SPLINE
SPL {X  -162.820, Y  +508.314, Z    +0.000, E1   +58.337, E3 +257283.169}
SPL {X  -162.820, Y  +498.518, Z    +0.000, E1   +58.346, E3 +257295.675}
SPL {X  -162.820, Y  +487.033, Z    +0.000, E1   +58.385, E3 +257310.273}
SPL {X  -162.820, Y  +474.470, Z    +0.000, E1   +58.318, E3 +257326.839}
SPL {X  -162.820, Y  +463.661, Z    +0.000, E1   +58.370, E3 +257340.278}
SPL {X  -162.820, Y  +454.904, Z    +0.000, E1   +58.380, E3 +257351.444}
SPL {X  -162.820, Y  +446.206, Z    +0.000, E1   +58.278, E3 +257363.335}
SPL {X  -162.820, Y  +436.416, Z    +0.000, E1   +58.325, E3 +257375.575}
SPL {X  -162.820, Y  +426.628, Z    +0.000, E1   +58.432, E3 +257387.443}
SPL {X  -162.820, Y  +415.377, Z    +0.000, E1   +58.239, E3 +257403.375}
SPL {X  -162.820, Y  +403.663, Z    +0.000, E1   +58.258, E3 +257418.154}
SPL {X  -162.820, Y  +397.157, Z    +0.000, E1   +58.054, E3 +257427.890}
SPL {X  -162.820, Y  +387.359, Z    +0.000, E1   +58.365, E3 +257438.519}
SPL {X  -162.810, Y  +378.731, Z    +0.000, E1   +58.366, E3 +257449.577}
SPL {X  -162.546, Y  +371.051, Z    +0.000, E1   +58.239, E3 +257460.297}
SPL {X  -161.863, Y  +362.875, Z    +0.000, E1   +58.273, E3 +257470.522}
SPL {X  -161.159, Y  +357.301, Z    +0.000, E1   +57.946, E3 +257479.822}
SPL {X  -159.864, Y  +349.614, Z    +0.000, E1   +57.922, E3 +257489.898}
SPL {X  -158.548, Y  +343.449, Z    +0.000, E1   +57.711, E3 +257499.072}
SPL {X  -156.580, Y  +335.856, Z    +0.000, E1   +57.340, E3 +257511.295}
SPL {X  -154.237, Y  +328.333, Z    +0.000, E1   +56.930, E3 +257523.214}
SPL {X  -152.732, Y  +324.078, Z    +0.000, E1   +56.482, E3 +257531.219}
SPL {X  -150.609, Y  +318.634, Z    +0.000, E1   +56.366, E3 +257538.913}
SPL {X  -148.206, Y  +313.080, Z    +0.000, E1   +55.888, E3 +257548.625}
SPL {X  -145.956, Y  +308.339, Z    +0.000, E1   +55.380, E3 +257557.301}
SPL {X  -143.330, Y  +303.254, Z    +0.000, E1   +55.057, E3 +257565.421}
SPL {X  -137.431, Y  +293.190, Z    +0.000, E1   +56.809, E3 +257569.584}
SPL {X  -115.845, Y  +266.087, Z    +0.000, E1   +50.276, E3 +257668.442}
SPL {X  -114.083, Y  +264.330, Z    +0.000, E1   +49.123, E3 +257707.152}
ENDSPLINE

SPLINE
SPL {X  -149.622, Y  +316.285, Z    +0.000, E1   +35.036, E3 +257775.664}
SPL {X  -158.704, Y  +344.121, Z    +0.000, E1   +23.312, E3 +257785.537}
SPL {X  -162.109, Y  +365.304, Z    +0.000, E1   +11.761, E3 +257784.839}
SPL {X  -162.811, Y  +378.776, Z    +0.000, E1    +3.078, E3 +257785.083}
SPL {X  -162.820, Y  +382.545, Z    +0.000, E1    +0.100, E3 +257784.644}
SPL {X  -162.820, Y  +384.317, Z    +0.000, E1    -1.618, E3 +257784.463}
SPL {X  -162.820, Y  +387.033, Z    +0.000, E1    -4.758, E3 +257784.255}
SPL {X  -162.820, Y  +390.967, Z    +0.000, E1    -9.918, E3 +257784.700}
SPL {X  -162.820, Y  +397.718, Z    +0.000, E1   -19.761, E3 +257784.074}
SPL {X  -162.820, Y  +405.058, Z    +0.000, E1   -29.962, E3 +257784.987}
SPL {X  -162.820, Y  +417.515, Z    +0.000, E1   -44.878, E3 +257784.149}
SPL {X  -162.820, Y  +462.065, Z    +0.000, E1   -61.507, E3 +257801.109}
SPL {X  -162.820, Y  +504.602, Z    +0.000, E1   -64.286, E3 +257826.635}
SPL {X  -162.820, Y  +535.709, Z    +0.000, E1   -59.182, E3 +257884.314}
SPL {X  -162.820, Y  +543.678, Z    +0.000, E1   -58.515, E3 +257898.703}
SPL {X  -162.820, Y  +553.725, Z    +0.000, E1   -58.454, E3 +257911.964}
SPL {X  -162.820, Y  +562.850, Z    +0.000, E1   -58.373, E3 +257924.126}
SPL {X  -162.820, Y  +571.217, Z    +0.000, E1   -58.397, E3 +257934.679}
SPL {X  -162.820, Y  +581.879, Z    +0.000, E1   -58.475, E3 +257947.932}
SPL {X  -162.820, Y  +591.768, Z    +0.000, E1   -58.375, E3 +257961.130}
SPL {X  -162.820, Y  +601.090, Z    +0.000, E1   -58.519, E3 +257972.117}
SPL {X  -162.820, Y  +609.492, Z    +0.000, E1   -58.431, E3 +257983.422}
SPL {X  -162.820, Y  +617.241, Z    +0.000, E1   -58.340, E3 +257993.947}
SPL {X  -162.820, Y  +626.506, Z    +0.000, E1   -58.420, E3 +258005.329}
SPL {X  -162.820, Y  +635.919, Z    +0.000, E1   -58.604, E3 +258016.073}
SPL {X  -162.820, Y  +643.895, Z    +0.000, E1   -58.380, E3 +258027.838}
SPL {X  -162.820, Y  +653.118, Z    +0.000, E1   -58.401, E3 +258039.435}
SPL {X  -162.820, Y  +660.924, Z    +0.000, E1   -58.393, E3 +258049.503}
SPL {X  -162.820, Y  +670.459, Z    +0.000, E1   -58.489, E3 +258061.104}
SPL {X  -162.713, Y  +679.396, Z    +0.000, E1   -58.414, E3 +258073.003}
SPL {X  -162.301, Y  +686.495, Z    +0.000, E1   -58.302, E3 +258082.787}
SPL {X  -161.571, Y  +693.631, Z    +0.000, E1   -58.186, E3 +258092.751}
SPL {X  -160.411, Y  +701.402, Z    +0.000, E1   -58.100, E3 +258103.227}
SPL {X  -159.229, Y  +707.508, Z    +0.000, E1   -57.870, E3 +258112.465}
SPL {X  -157.825, Y  +713.519, Z    +0.000, E1   -57.630, E3 +258121.701}
SPL {X  -156.079, Y  +719.864, Z    +0.000, E1   -57.324, E3 +258131.664}
SPL {X  -154.064, Y  +726.175, Z    +0.000, E1   -57.042, E3 +258141.426}
SPL {X  -152.053, Y  +731.726, Z    +0.000, E1   -56.648, E3 +258150.711}
SPL {X  -150.108, Y  +736.570, Z    +0.000, E1   -56.283, E3 +258158.950}
SPL {X  -147.726, Y  +741.964, Z    +0.000, E1   -55.884, E3 +258167.986}
SPL {X  -145.163, Y  +747.242, Z    +0.000, E1   -55.517, E3 +258176.582}
SPL {X  -142.489, Y  +752.286, Z    +0.000, E1   -55.227, E3 +258184.409}
SPL {X  -136.074, Y  +762.910, Z    +0.000, E1   -57.336, E3 +258187.531}
SPL {X  -116.561, Y  +787.183, Z    +0.000, E1   -51.088, E3 +258271.999}
ENDSPLINE

SPLINE
SPL {X  -119.623, Y  +783.957, Z    +0.000, E1   -49.202, E3 +258396.532}
SPL {X  -149.958, Y  +736.927, Z    +0.000, E1   -34.772, E3 +258394.249}
SPL {X  -158.826, Y  +709.343, Z    +0.000, E1   -23.029, E3 +258402.592}
SPL {X  -161.800, Y  +691.694, Z    +0.000, E1   -13.520, E3 +258404.886}
SPL {X  -162.711, Y  +679.444, Z    +0.000, E1    -5.922, E3 +258404.960}
SPL {X  -162.820, Y  +673.886, Z    +0.000, E1    -1.998, E3 +258405.121}
SPL {X  -162.820, Y  +671.620, Z    +0.000, E1    -0.225, E3 +258404.696}
SPL {X  -162.820, Y  +669.030, Z    +0.000, E1    +2.242, E3 +258404.397}
SPL {X  -162.820, Y  +664.667, Z    +0.000, E1    +7.867, E3 +258404.100}
SPL {X  -162.820, Y  +660.022, Z    +0.000, E1   +14.535, E3 +258403.997}
SPL {X  -162.820, Y  +653.408, Z    +0.000, E1   +24.221, E3 +258404.307}
SPL {X  -162.820, Y  +640.244, Z    +0.000, E1   +41.042, E3 +258404.351}
SPL {X  -162.820, Y  +592.517, Z    +0.000, E1   +60.575, E3 +258423.482}
SPL {X  -162.820, Y  +515.613, Z    +0.000, E1   +60.751, E3 +258497.317}
ENDSPLINE

SPLINE
SPL {X  -162.820, Y  +518.198, Z    +0.000, E1   +58.338, E3 +258510.473}
ENDSPLINE

SPLINE
SPL {X  -162.820, Y  +508.314, Z    +0.000, E1   +58.337, E3 +258523.169}
SPL {X  -162.820, Y  +498.518, Z    +0.000, E1   +58.346, E3 +258535.675}
SPL {X  -162.820, Y  +489.418, Z    +0.000, E1   +58.357, E3 +258547.265}
SPL {X  -162.820, Y  +479.904, Z    +0.000, E1   +58.389, E3 +258559.312}
SPL {X  -162.820, Y  +472.095, Z    +0.000, E1   +58.202, E3 +258570.492}
SPL {X  -162.820, Y  +463.661, Z    +0.000, E1   +58.370, E3 +258580.278}
SPL {X  -162.820, Y  +454.904, Z    +0.000, E1   +58.380, E3 +258591.444}
SPL {X  -162.820, Y  +446.206, Z    +0.000, E1   +58.278, E3 +258603.335}
SPL {X  -162.820, Y  +436.416, Z    +0.000, E1   +58.325, E3 +258615.575}
SPL {X  -162.820, Y  +426.628, Z    +0.000, E1   +58.432, E3 +258627.443}
SPL {X  -162.820, Y  +418.389, Z    +0.000, E1   +58.300, E3 +258638.846}
SPL {X  -162.820, Y  +412.292, Z    +0.000, E1   +58.070, E3 +258648.214}
SPL {X  -162.820, Y  +403.663, Z    +0.000, E1   +58.258, E3 +258658.154}
SPL {X  -162.820, Y  +397.157, Z    +0.000, E1   +58.054, E3 +258667.890}
SPL {X  -162.820, Y  +387.359, Z    +0.000, E1   +58.365, E3 +258678.519}
SPL {X  -162.810, Y  +378.731, Z    +0.000, E1   +58.366, E3 +258689.577}
SPL {X  -162.546, Y  +371.051, Z    +0.000, E1   +58.239, E3 +258700.297}
SPL {X  -161.863, Y  +362.875, Z    +0.000, E1   +58.273, E3 +258710.522}
SPL {X  -161.159, Y  +357.301, Z    +0.000, E1   +57.946, E3 +258719.822}
SPL {X  -159.864, Y  +349.614, Z    +0.000, E1   +57.922, E3 +258729.898}
SPL {X  -158.548, Y  +343.449, Z    +0.000, E1   +57.711, E3 +258739.072}
SPL {X  -156.580, Y  +335.856, Z    +0.000, E1   +57.340, E3 +258751.295}
SPL {X  -154.237, Y  +328.333, Z    +0.000, E1   +56.930, E3 +258763.214}
SPL {X  -152.732, Y  +324.078, Z    +0.000, E1   +56.482, E3 +258771.219}
SPL {X  -150.609, Y  +318.634, Z    +0.000, E1   +56.366, E3 +258778.913}
SPL {X  -148.206, Y  +313.080, Z    +0.000, E1   +55.888, E3 +258788.625}
SPL {X  -145.956, Y  +308.339, Z    +0.000, E1   +55.380, E3 +258797.301}
SPL {X  -143.330, Y  +303.254, Z    +0.000, E1   +55.057, E3 +258805.421}
SPL {X  -137.431, Y  +293.190, Z    +0.000, E1   +56.809, E3 +258809.584}
SPL {X  -115.845, Y  +266.087, Z    +0.000, E1   +50.276, E3 +258908.442}
SPL {X  -114.083, Y  +264.330, Z    +0.000, E1   +49.123, E3 +258947.152}
ENDSPLINE

SPLINE
SPL {X  -149.622, Y  +316.285, Z    +0.000, E1   +35.036, E3 +259015.664}
SPL {X  -158.704, Y  +344.121, Z    +0.000, E1   +23.312, E3 +259025.537}
SPL {X  -162.109, Y  +365.304, Z    +0.000, E1   +11.761, E3 +259024.839}
SPL {X  -162.811, Y  +378.776, Z    +0.000, E1    +3.078, E3 +259025.083}
SPL {X  -162.820, Y  +383.454, Z    +0.000, E1    -0.619, E3 +259024.551}
SPL {X  -162.820, Y  +387.033, Z    +0.000, E1    -4.758, E3 +259024.255}
SPL {X  -162.820, Y  +390.967, Z    +0.000, E1    -9.918, E3 +259024.700}
SPL {X  -162.820, Y  +397.718, Z    +0.000, E1   -19.761, E3 +259024.074}
SPL {X  -162.820, Y  +405.058, Z    +0.000, E1   -29.962, E3 +259024.987}
SPL {X  -162.820, Y  +417.515, Z    +0.000, E1   -44.878, E3 +259024.149}
SPL {X  -162.820, Y  +462.065, Z    +0.000, E1   -61.507, E3 +259041.109}
SPL {X  -162.820, Y  +504.602, Z    +0.000, E1   -64.286, E3 +259066.635}
SPL {X  -162.820, Y  +535.709, Z    +0.000, E1   -59.182, E3 +259124.314}
SPL {X  -162.820, Y  +543.678, Z    +0.000, E1   -58.515, E3 +259138.703}
SPL {X  -162.820, Y  +553.725, Z    +0.000, E1   -58.454, E3 +259151.964}
SPL {X  -162.820, Y  +562.850, Z    +0.000, E1   -58.373, E3 +259164.126}
SPL {X  -162.820, Y  +573.452, Z    +0.000, E1   -58.444, E3 +259177.339}
SPL {X  -162.820, Y  +583.632, Z    +0.000, E1   -58.444, E3 +259190.266}
SPL {X  -162.820, Y  +591.768, Z    +0.000, E1   -58.375, E3 +259201.130}
SPL {X  -162.820, Y  +601.090, Z    +0.000, E1   -58.519, E3 +259212.117}
SPL {X  -162.820, Y  +609.492, Z    +0.000, E1   -58.431, E3 +259223.422}
SPL {X  -162.820, Y  +617.241, Z    +0.000, E1   -58.340, E3 +259233.947}
SPL {X  -162.820, Y  +626.506, Z    +0.000, E1   -58.420, E3 +259245.329}
SPL {X  -162.820, Y  +635.919, Z    +0.000, E1   -58.604, E3 +259256.073}
SPL {X  -162.820, Y  +643.895, Z    +0.000, E1   -58.380, E3 +259267.838}
SPL {X  -162.820, Y  +653.118, Z    +0.000, E1   -58.401, E3 +259279.435}
SPL {X  -162.820, Y  +660.924, Z    +0.000, E1   -58.393, E3 +259289.503}
SPL {X  -162.820, Y  +670.459, Z    +0.000, E1   -58.489, E3 +259301.104}
SPL {X  -162.713, Y  +679.396, Z    +0.000, E1   -58.414, E3 +259313.003}
SPL {X  -162.301, Y  +686.495, Z    +0.000, E1   -58.302, E3 +259322.787}
SPL {X  -161.571, Y  +693.631, Z    +0.000, E1   -58.186, E3 +259332.751}
SPL {X  -160.411, Y  +701.402, Z    +0.000, E1   -58.100, E3 +259343.227}
SPL {X  -159.229, Y  +707.508, Z    +0.000, E1   -57.870, E3 +259352.465}
SPL {X  -157.825, Y  +713.519, Z    +0.000, E1   -57.630, E3 +259361.701}
SPL {X  -156.079, Y  +719.864, Z    +0.000, E1   -57.324, E3 +259371.664}
SPL {X  -154.064, Y  +726.175, Z    +0.000, E1   -57.042, E3 +259381.426}
SPL {X  -152.053, Y  +731.726, Z    +0.000, E1   -56.648, E3 +259390.711}
SPL {X  -150.108, Y  +736.570, Z    +0.000, E1   -56.283, E3 +259398.950}
SPL {X  -147.726, Y  +741.964, Z    +0.000, E1   -55.884, E3 +259407.986}
SPL {X  -145.163, Y  +747.242, Z    +0.000, E1   -55.517, E3 +259416.582}
SPL {X  -142.489, Y  +752.286, Z    +0.000, E1   -55.227, E3 +259424.409}
SPL {X  -136.074, Y  +762.910, Z    +0.000, E1   -57.336, E3 +259427.531}
SPL {X  -116.561, Y  +787.183, Z    +0.000, E1   -51.088, E3 +259511.999}
ENDSPLINE

SPLINE
SPL {X  -119.623, Y  +783.957, Z    +0.000, E1   -49.202, E3 +259636.532}
SPL {X  -149.958, Y  +736.927, Z    +0.000, E1   -34.772, E3 +259634.249}
SPL {X  -158.826, Y  +709.343, Z    +0.000, E1   -23.029, E3 +259642.592}
SPL {X  -161.800, Y  +691.694, Z    +0.000, E1   -13.520, E3 +259644.886}
SPL {X  -162.711, Y  +679.444, Z    +0.000, E1    -5.922, E3 +259644.960}
SPL {X  -162.820, Y  +672.303, Z    +0.000, E1    -0.875, E3 +259644.825}
SPL {X  -162.820, Y  +669.030, Z    +0.000, E1    +2.242, E3 +259644.397}
SPL {X  -162.820, Y  +664.667, Z    +0.000, E1    +7.867, E3 +259644.100}
SPL {X  -162.820, Y  +660.022, Z    +0.000, E1   +14.535, E3 +259643.997}
SPL {X  -162.820, Y  +653.408, Z    +0.000, E1   +24.221, E3 +259644.307}
SPL {X  -162.820, Y  +640.244, Z    +0.000, E1   +41.042, E3 +259644.351}
SPL {X  -162.820, Y  +592.517, Z    +0.000, E1   +60.575, E3 +259663.482}
SPL {X  -162.820, Y  +515.613, Z    +0.000, E1   +60.751, E3 +259737.317}
ENDSPLINE

SPLINE
SPL {X  -162.820, Y  +518.198, Z    +0.000, E1   +58.338, E3 +259750.473}
ENDSPLINE

SPLINE
SPL {X  -162.820, Y  +508.314, Z    +0.000, E1   +58.337, E3 +259763.169}
SPL {X  -162.820, Y  +498.518, Z    +0.000, E1   +58.346, E3 +259775.675}
SPL {X  -162.820, Y  +489.418, Z    +0.000, E1   +58.357, E3 +259787.265}
SPL {X  -162.820, Y  +479.904, Z    +0.000, E1   +58.389, E3 +259799.312}
SPL {X  -162.820, Y  +472.095, Z    +0.000, E1   +58.202, E3 +259810.492}
SPL {X  -162.820, Y  +463.661, Z    +0.000, E1   +58.370, E3 +259820.278}
SPL {X  -162.820, Y  +454.904, Z    +0.000, E1   +58.380, E3 +259831.444}
SPL {X  -162.820, Y  +446.206, Z    +0.000, E1   +58.278, E3 +259843.335}
SPL {X  -162.820, Y  +436.416, Z    +0.000, E1   +58.325, E3 +259855.575}
SPL {X  -162.820, Y  +426.628, Z    +0.000, E1   +58.432, E3 +259867.443}
SPL {X  -162.820, Y  +415.377, Z    +0.000, E1   +58.239, E3 +259883.375}
SPL {X  -162.820, Y  +403.663, Z    +0.000, E1   +58.258, E3 +259898.154}
SPL {X  -162.820, Y  +397.157, Z    +0.000, E1   +58.054, E3 +259907.890}
SPL {X  -162.820, Y  +387.359, Z    +0.000, E1   +58.365, E3 +259918.519}
SPL {X  -162.810, Y  +378.731, Z    +0.000, E1   +58.366, E3 +259929.577}
SPL {X  -162.546, Y  +371.051, Z    +0.000, E1   +58.239, E3 +259940.297}
SPL {X  -161.863, Y  +362.875, Z    +0.000, E1   +58.273, E3 +259950.522}
SPL {X  -161.159, Y  +357.301, Z    +0.000, E1   +57.946, E3 +259959.822}
SPL {X  -159.864, Y  +349.614, Z    +0.000, E1   +57.922, E3 +259969.898}
SPL {X  -158.548, Y  +343.449, Z    +0.000, E1   +57.711, E3 +259979.072}
SPL {X  -156.580, Y  +335.856, Z    +0.000, E1   +57.340, E3 +259991.295}
SPL {X  -154.237, Y  +328.333, Z    +0.000, E1   +56.930, E3 +260003.214}
SPL {X  -152.732, Y  +324.078, Z    +0.000, E1   +56.482, E3 +260011.219}
SPL {X  -150.609, Y  +318.634, Z    +0.000, E1   +56.366, E3 +260018.913}
SPL {X  -148.206, Y  +313.080, Z    +0.000, E1   +55.888, E3 +260028.625}
SPL {X  -145.956, Y  +308.339, Z    +0.000, E1   +55.380, E3 +260037.301}
SPL {X  -143.330, Y  +303.254, Z    +0.000, E1   +55.057, E3 +260045.421}
SPL {X  -137.431, Y  +293.190, Z    +0.000, E1   +56.809, E3 +260049.584}
SPL {X  -115.845, Y  +266.087, Z    +0.000, E1   +50.276, E3 +260148.442}
SPL {X  -114.083, Y  +264.330, Z    +0.000, E1   +49.123, E3 +260187.152}
ENDSPLINE

SPLINE
SPL {X  -149.622, Y  +316.285, Z    +0.000, E1   +35.036, E3 +260255.664}
SPL {X  -158.704, Y  +344.121, Z    +0.000, E1   +23.312, E3 +260265.537}
SPL {X  -161.701, Y  +361.440, Z    +0.000, E1   +13.961, E3 +260264.608}
SPL {X  -162.691, Y  +374.019, Z    +0.000, E1    +6.263, E3 +260265.261}
SPL {X  -162.820, Y  +381.771, Z    +0.000, E1    +0.850, E3 +260264.745}
SPL {X  -162.820, Y  +384.317, Z    +0.000, E1    -1.618, E3 +260264.463}
SPL {X  -162.820, Y  +387.033, Z    +0.000, E1    -4.758, E3 +260264.255}
SPL {X  -162.820, Y  +390.967, Z    +0.000, E1    -9.918, E3 +260264.700}
SPL {X  -162.820, Y  +395.392, Z    +0.000, E1   -16.726, E3 +260263.141}
SPL {X  -162.820, Y  +402.654, Z    +0.000, E1   -26.492, E3 +260265.032}
SPL {X  -162.820, Y  +417.515, Z    +0.000, E1   -44.878, E3 +260264.149}
SPL {X  -162.820, Y  +462.065, Z    +0.000, E1   -61.507, E3 +260281.109}
SPL {X  -162.820, Y  +504.602, Z    +0.000, E1   -64.286, E3 +260306.635}
SPL {X  -162.820, Y  +535.709, Z    +0.000, E1   -59.182, E3 +260364.314}
SPL {X  -162.820, Y  +543.678, Z    +0.000, E1   -58.515, E3 +260378.703}
SPL {X  -162.820, Y  +553.725, Z    +0.000, E1   -58.454, E3 +260391.964}
SPL {X  -162.820, Y  +562.850, Z    +0.000, E1   -58.373, E3 +260404.126}
SPL {X  -162.820, Y  +571.217, Z    +0.000, E1   -58.397, E3 +260414.679}
SPL {X  -162.820, Y  +581.879, Z    +0.000, E1   -58.475, E3 +260427.932}
SPL {X  -162.820, Y  +591.768, Z    +0.000, E1   -58.375, E3 +260441.130}
SPL {X  -162.820, Y  +601.090, Z    +0.000, E1   -58.519, E3 +260452.117}
SPL {X  -162.820, Y  +609.492, Z    +0.000, E1   -58.431, E3 +260463.422}
SPL {X  -162.820, Y  +617.241, Z    +0.000, E1   -58.340, E3 +260473.947}
SPL {X  -162.820, Y  +626.506, Z    +0.000, E1   -58.420, E3 +260485.329}
SPL {X  -162.820, Y  +635.919, Z    +0.000, E1   -58.604, E3 +260496.073}
SPL {X  -162.820, Y  +643.895, Z    +0.000, E1   -58.380, E3 +260507.838}
SPL {X  -162.820, Y  +653.118, Z    +0.000, E1   -58.401, E3 +260519.435}
SPL {X  -162.820, Y  +660.924, Z    +0.000, E1   -58.393, E3 +260529.503}
SPL {X  -162.820, Y  +670.459, Z    +0.000, E1   -58.489, E3 +260541.104}
SPL {X  -162.713, Y  +679.396, Z    +0.000, E1   -58.414, E3 +260553.003}
SPL {X  -162.301, Y  +686.495, Z    +0.000, E1   -58.302, E3 +260562.787}
SPL {X  -161.571, Y  +693.631, Z    +0.000, E1   -58.186, E3 +260572.751}
SPL {X  -160.411, Y  +701.402, Z    +0.000, E1   -58.100, E3 +260583.227}
SPL {X  -159.229, Y  +707.508, Z    +0.000, E1   -57.870, E3 +260592.465}
SPL {X  -157.825, Y  +713.519, Z    +0.000, E1   -57.630, E3 +260601.701}
SPL {X  -156.079, Y  +719.864, Z    +0.000, E1   -57.324, E3 +260611.664}
SPL {X  -154.064, Y  +726.175, Z    +0.000, E1   -57.042, E3 +260621.426}
SPL {X  -152.053, Y  +731.726, Z    +0.000, E1   -56.648, E3 +260630.711}
SPL {X  -150.108, Y  +736.570, Z    +0.000, E1   -56.283, E3 +260638.950}
SPL {X  -147.726, Y  +741.964, Z    +0.000, E1   -55.884, E3 +260647.986}
SPL {X  -145.163, Y  +747.242, Z    +0.000, E1   -55.517, E3 +260656.582}
SPL {X  -142.489, Y  +752.286, Z    +0.000, E1   -55.227, E3 +260664.409}
SPL {X  -136.074, Y  +762.910, Z    +0.000, E1   -57.336, E3 +260667.531}
SPL {X  -116.561, Y  +787.183, Z    +0.000, E1   -51.088, E3 +260751.999}
ENDSPLINE

SPLINE
SPL {X  -119.623, Y  +783.957, Z    +0.000, E1   -49.202, E3 +260876.532}
SPL {X  -149.958, Y  +736.927, Z    +0.000, E1   -34.772, E3 +260874.249}
SPL {X  -158.826, Y  +709.343, Z    +0.000, E1   -23.029, E3 +260882.592}
SPL {X  -161.800, Y  +691.694, Z    +0.000, E1   -13.520, E3 +260884.886}
SPL {X  -162.711, Y  +679.444, Z    +0.000, E1    -5.922, E3 +260884.960}
SPL {X  -162.820, Y  +672.303, Z    +0.000, E1    -0.875, E3 +260884.825}
SPL {X  -162.820, Y  +669.030, Z    +0.000, E1    +2.242, E3 +260884.397}
SPL {X  -162.820, Y  +664.667, Z    +0.000, E1    +7.867, E3 +260884.100}
SPL {X  -162.820, Y  +660.022, Z    +0.000, E1   +14.535, E3 +260883.997}
SPL {X  -162.820, Y  +653.408, Z    +0.000, E1   +24.221, E3 +260884.307}
SPL {X  -162.820, Y  +640.244, Z    +0.000, E1   +41.042, E3 +260884.351}
SPL {X  -162.820, Y  +602.578, Z    +0.000, E1   +60.061, E3 +260895.766}
SPL {X  -162.820, Y  +586.468, Z    +0.000, E1   +60.779, E3 +260908.168}
SPL {X  -162.820, Y  +515.613, Z    +0.000, E1   +60.751, E3 +260977.317}
ENDSPLINE

SPLINE
SPL {X  -162.820, Y  +518.198, Z    +0.000, E1   +58.338, E3 +260990.473}
ENDSPLINE

SPLINE
SPL {X  -162.820, Y  +508.314, Z    +0.000, E1   +58.337, E3 +261003.169}
SPL {X  -162.820, Y  +498.518, Z    +0.000, E1   +58.346, E3 +261015.675}
SPL {X  -162.820, Y  +489.418, Z    +0.000, E1   +58.357, E3 +261027.265}
SPL {X  -162.820, Y  +479.904, Z    +0.000, E1   +58.389, E3 +261039.312}
SPL {X  -162.820, Y  +472.095, Z    +0.000, E1   +58.202, E3 +261050.492}
SPL {X  -162.820, Y  +463.661, Z    +0.000, E1   +58.370, E3 +261060.278}
SPL {X  -162.820, Y  +454.904, Z    +0.000, E1   +58.380, E3 +261071.444}
SPL {X  -162.820, Y  +446.206, Z    +0.000, E1   +58.278, E3 +261083.335}
SPL {X  -162.820, Y  +436.416, Z    +0.000, E1   +58.325, E3 +261095.575}
SPL {X  -162.820, Y  +426.628, Z    +0.000, E1   +58.432, E3 +261107.443}
SPL {X  -162.820, Y  +415.377, Z    +0.000, E1   +58.239, E3 +261123.375}
SPL {X  -162.820, Y  +403.663, Z    +0.000, E1   +58.258, E3 +261138.154}
SPL {X  -162.820, Y  +397.157, Z    +0.000, E1   +58.054, E3 +261147.890}
SPL {X  -162.820, Y  +387.359, Z    +0.000, E1   +58.365, E3 +261158.519}
SPL {X  -162.810, Y  +378.731, Z    +0.000, E1   +58.366, E3 +261169.577}
SPL {X  -162.546, Y  +371.051, Z    +0.000, E1   +58.239, E3 +261180.297}
SPL {X  -161.863, Y  +362.875, Z    +0.000, E1   +58.273, E3 +261190.522}
SPL {X  -161.159, Y  +357.301, Z    +0.000, E1   +57.946, E3 +261199.822}
SPL {X  -159.864, Y  +349.614, Z    +0.000, E1   +57.922, E3 +261209.898}
SPL {X  -158.548, Y  +343.449, Z    +0.000, E1   +57.711, E3 +261219.072}
SPL {X  -156.580, Y  +335.856, Z    +0.000, E1   +57.340, E3 +261231.295}
SPL {X  -154.237, Y  +328.333, Z    +0.000, E1   +56.930, E3 +261243.214}
SPL {X  -152.732, Y  +324.078, Z    +0.000, E1   +56.482, E3 +261251.219}
SPL {X  -150.609, Y  +318.634, Z    +0.000, E1   +56.366, E3 +261258.913}
SPL {X  -148.206, Y  +313.080, Z    +0.000, E1   +55.888, E3 +261268.625}
SPL {X  -145.956, Y  +308.339, Z    +0.000, E1   +55.380, E3 +261277.301}
SPL {X  -143.330, Y  +303.254, Z    +0.000, E1   +55.057, E3 +261285.421}
SPL {X  -137.431, Y  +293.190, Z    +0.000, E1   +56.809, E3 +261289.584}
SPL {X  -115.845, Y  +266.087, Z    +0.000, E1   +50.276, E3 +261388.442}
SPL {X  -114.083, Y  +264.330, Z    +0.000, E1   +49.123, E3 +261427.152}
ENDSPLINE

SPLINE
SPL {X  -136.188, Y  +291.263, Z    +0.000, E1   +45.457, E3 +261523.218}
SPL {X  -151.738, Y  +321.457, Z    +0.000, E1   +32.773, E3 +261490.387}
SPL {X  -158.704, Y  +344.121, Z    +0.000, E1   +23.312, E3 +261505.537}
SPL {X  -161.701, Y  +361.440, Z    +0.000, E1   +13.961, E3 +261504.608}
SPL {X  -162.691, Y  +374.019, Z    +0.000, E1    +6.263, E3 +261505.261}
SPL {X  -162.820, Y  +380.238, Z    +0.000, E1    +1.925, E3 +261504.945}
SPL {X  -162.820, Y  +382.545, Z    +0.000, E1    +0.100, E3 +261504.644}
SPL {X  -162.820, Y  +384.317, Z    +0.000, E1    -1.618, E3 +261504.463}
SPL {X  -162.820, Y  +387.033, Z    +0.000, E1    -4.758, E3 +261504.255}
SPL {X  -162.820, Y  +390.967, Z    +0.000, E1    -9.918, E3 +261504.700}
SPL {X  -162.820, Y  +395.392, Z    +0.000, E1   -16.726, E3 +261503.141}
SPL {X  -162.820, Y  +402.654, Z    +0.000, E1   -26.492, E3 +261505.032}
SPL {X  -162.820, Y  +417.515, Z    +0.000, E1   -44.878, E3 +261504.149}
SPL {X  -162.820, Y  +462.065, Z    +0.000, E1   -61.507, E3 +261521.109}
SPL {X  -162.820, Y  +504.602, Z    +0.000, E1   -64.286, E3 +261546.635}
SPL {X  -162.820, Y  +535.709, Z    +0.000, E1   -59.182, E3 +261604.314}
SPL {X  -162.820, Y  +543.678, Z    +0.000, E1   -58.515, E3 +261618.703}
SPL {X  -162.820, Y  +553.725, Z    +0.000, E1   -58.454, E3 +261631.964}
SPL {X  -162.820, Y  +562.850, Z    +0.000, E1   -58.373, E3 +261644.126}
SPL {X  -162.820, Y  +573.452, Z    +0.000, E1   -58.444, E3 +261657.339}
SPL {X  -162.820, Y  +583.632, Z    +0.000, E1   -58.444, E3 +261670.266}
SPL {X  -162.820, Y  +591.768, Z    +0.000, E1   -58.375, E3 +261681.130}
SPL {X  -162.820, Y  +601.090, Z    +0.000, E1   -58.519, E3 +261692.117}
SPL {X  -162.820, Y  +609.492, Z    +0.000, E1   -58.431, E3 +261703.422}
SPL {X  -162.820, Y  +617.241, Z    +0.000, E1   -58.340, E3 +261713.947}
SPL {X  -162.820, Y  +626.506, Z    +0.000, E1   -58.420, E3 +261725.329}
SPL {X  -162.820, Y  +638.850, Z    +0.000, E1   -58.527, E3 +261740.545}
SPL {X  -162.820, Y  +651.112, Z    +0.000, E1   -58.411, E3 +261756.903}
SPL {X  -162.820, Y  +660.924, Z    +0.000, E1   -58.393, E3 +261769.503}
SPL {X  -162.820, Y  +670.459, Z    +0.000, E1   -58.489, E3 +261781.104}
SPL {X  -162.713, Y  +679.396, Z    +0.000, E1   -58.414, E3 +261793.003}
SPL {X  -162.301, Y  +686.495, Z    +0.000, E1   -58.302, E3 +261802.787}
SPL {X  -161.571, Y  +693.631, Z    +0.000, E1   -58.186, E3 +261812.751}
SPL {X  -160.411, Y  +701.402, Z    +0.000, E1   -58.100, E3 +261823.227}
SPL {X  -159.229, Y  +707.508, Z    +0.000, E1   -57.870, E3 +261832.465}
SPL {X  -157.825, Y  +713.519, Z    +0.000, E1   -57.630, E3 +261841.701}
SPL {X  -156.079, Y  +719.864, Z    +0.000, E1   -57.324, E3 +261851.664}
SPL {X  -154.064, Y  +726.175, Z    +0.000, E1   -57.042, E3 +261861.426}
SPL {X  -152.053, Y  +731.726, Z    +0.000, E1   -56.648, E3 +261870.711}
SPL {X  -150.108, Y  +736.570, Z    +0.000, E1   -56.283, E3 +261878.950}
SPL {X  -147.726, Y  +741.964, Z    +0.000, E1   -55.884, E3 +261887.986}
SPL {X  -145.163, Y  +747.242, Z    +0.000, E1   -55.517, E3 +261896.582}
SPL {X  -142.489, Y  +752.286, Z    +0.000, E1   -55.227, E3 +261904.409}
SPL {X  -136.074, Y  +762.910, Z    +0.000, E1   -57.336, E3 +261907.531}
SPL {X  -116.561, Y  +787.183, Z    +0.000, E1   -51.088, E3 +261991.999}
ENDSPLINE

SPLINE
SPL {X  -119.623, Y  +783.957, Z    +0.000, E1   -49.202, E3 +262116.532}
SPL {X  -149.958, Y  +736.927, Z    +0.000, E1   -34.772, E3 +262114.249}
SPL {X  -158.826, Y  +709.343, Z    +0.000, E1   -23.029, E3 +262122.592}
SPL {X  -161.800, Y  +691.694, Z    +0.000, E1   -13.520, E3 +262124.886}
SPL {X  -162.597, Y  +682.022, Z    +0.000, E1    -7.544, E3 +262124.542}
SPL {X  -162.813, Y  +675.055, Z    +0.000, E1    -2.911, E3 +262125.184}
SPL {X  -162.820, Y  +671.620, Z    +0.000, E1    -0.225, E3 +262124.696}
SPL {X  -162.820, Y  +669.030, Z    +0.000, E1    +2.242, E3 +262124.397}
SPL {X  -162.820, Y  +664.667, Z    +0.000, E1    +7.867, E3 +262124.100}
SPL {X  -162.820, Y  +660.022, Z    +0.000, E1   +14.535, E3 +262123.997}
SPL {X  -162.820, Y  +653.408, Z    +0.000, E1   +24.221, E3 +262124.307}
SPL {X  -162.820, Y  +640.244, Z    +0.000, E1   +41.042, E3 +262124.351}
SPL {X  -162.820, Y  +592.517, Z    +0.000, E1   +60.575, E3 +262143.482}
SPL {X  -162.820, Y  +515.613, Z    +0.000, E1   +60.751, E3 +262217.317}
ENDSPLINE

SPLINE
SPL {X  -162.820, Y  +518.198, Z    +0.000, E1   +58.338, E3 +262230.473}
ENDSPLINE

SPLINE
SPL {X  -162.820, Y  +508.314, Z    +0.000, E1   +58.337, E3 +262243.169}
SPL {X  -162.820, Y  +498.518, Z    +0.000, E1   +58.346, E3 +262255.675}
SPL {X  -162.820, Y  +489.418, Z    +0.000, E1   +58.357, E3 +262267.265}
SPL {X  -162.820, Y  +479.904, Z    +0.000, E1   +58.389, E3 +262279.312}
SPL {X  -162.820, Y  +472.095, Z    +0.000, E1   +58.202, E3 +262290.492}
SPL {X  -162.820, Y  +463.661, Z    +0.000, E1   +58.370, E3 +262300.278}
SPL {X  -162.820, Y  +454.904, Z    +0.000, E1   +58.380, E3 +262311.444}
SPL {X  -162.820, Y  +446.206, Z    +0.000, E1   +58.278, E3 +262323.335}
SPL {X  -162.820, Y  +436.416, Z    +0.000, E1   +58.325, E3 +262335.575}
SPL {X  -162.820, Y  +426.628, Z    +0.000, E1   +58.432, E3 +262347.443}
SPL {X  -162.820, Y  +415.377, Z    +0.000, E1   +58.239, E3 +262363.375}
SPL {X  -162.820, Y  +403.663, Z    +0.000, E1   +58.258, E3 +262378.154}
SPL {X  -162.820, Y  +397.157, Z    +0.000, E1   +58.054, E3 +262387.890}
SPL {X  -162.820, Y  +387.359, Z    +0.000, E1   +58.365, E3 +262398.519}
SPL {X  -162.810, Y  +378.731, Z    +0.000, E1   +58.366, E3 +262409.577}
SPL {X  -162.546, Y  +371.051, Z    +0.000, E1   +58.239, E3 +262420.297}
SPL {X  -161.863, Y  +362.875, Z    +0.000, E1   +58.273, E3 +262430.522}
SPL {X  -161.159, Y  +357.301, Z    +0.000, E1   +57.946, E3 +262439.822}
SPL {X  -159.864, Y  +349.614, Z    +0.000, E1   +57.922, E3 +262449.898}
SPL {X  -158.300, Y  +342.404, Z    +0.000, E1   +57.579, E3 +262461.344}
SPL {X  -156.187, Y  +334.499, Z    +0.000, E1   +57.331, E3 +262473.004}
SPL {X  -154.237, Y  +328.333, Z    +0.000, E1   +56.930, E3 +262483.214}
SPL {X  -152.732, Y  +324.078, Z    +0.000, E1   +56.482, E3 +262491.219}
SPL {X  -150.609, Y  +318.634, Z    +0.000, E1   +56.366, E3 +262498.913}
SPL {X  -148.206, Y  +313.080, Z    +0.000, E1   +55.888, E3 +262508.625}
SPL {X  -145.956, Y  +308.339, Z    +0.000, E1   +55.380, E3 +262517.301}
SPL {X  -142.234, Y  +301.255, Z    +0.000, E1   +55.418, E3 +262526.175}
SPL {X  -134.491, Y  +288.726, Z    +0.000, E1   +57.448, E3 +262531.831}
SPL {X  -115.845, Y  +266.087, Z    +0.000, E1   +50.276, E3 +262628.442}
SPL {X  -114.083, Y  +264.330, Z    +0.000, E1   +49.123, E3 +262667.152}
ENDSPLINE

SPLINE
SPL {X  -136.188, Y  +291.263, Z    +0.000, E1   +45.457, E3 +262763.218}
SPL {X  -151.738, Y  +321.457, Z    +0.000, E1   +32.773, E3 +262730.387}
SPL {X  -158.704, Y  +344.121, Z    +0.000, E1   +23.312, E3 +262745.537}
SPL {X  -162.109, Y  +365.304, Z    +0.000, E1   +11.761, E3 +262744.839}
SPL {X  -162.811, Y  +378.776, Z    +0.000, E1    +3.078, E3 +262745.083}
SPL {X  -162.820, Y  +382.545, Z    +0.000, E1    +0.100, E3 +262744.644}
SPL {X  -162.820, Y  +384.317, Z    +0.000, E1    -1.618, E3 +262744.463}
SPL {X  -162.820, Y  +387.033, Z    +0.000, E1    -4.758, E3 +262744.255}
SPL {X  -162.820, Y  +390.967, Z    +0.000, E1    -9.918, E3 +262744.700}
SPL {X  -162.820, Y  +395.392, Z    +0.000, E1   -16.726, E3 +262743.141}
SPL {X  -162.820, Y  +402.654, Z    +0.000, E1   -26.492, E3 +262745.032}
SPL {X  -162.820, Y  +417.515, Z    +0.000, E1   -44.878, E3 +262744.149}
SPL {X  -162.820, Y  +462.065, Z    +0.000, E1   -61.507, E3 +262761.109}
SPL {X  -162.820, Y  +504.602, Z    +0.000, E1   -64.286, E3 +262786.635}
SPL {X  -162.820, Y  +535.709, Z    +0.000, E1   -59.182, E3 +262844.314}
SPL {X  -162.820, Y  +543.678, Z    +0.000, E1   -58.515, E3 +262858.703}
SPL {X  -162.820, Y  +553.725, Z    +0.000, E1   -58.454, E3 +262871.964}
SPL {X  -162.820, Y  +562.850, Z    +0.000, E1   -58.373, E3 +262884.126}
SPL {X  -162.820, Y  +573.452, Z    +0.000, E1   -58.444, E3 +262897.339}
SPL {X  -162.820, Y  +583.632, Z    +0.000, E1   -58.444, E3 +262910.266}
SPL {X  -162.820, Y  +591.768, Z    +0.000, E1   -58.375, E3 +262921.130}
SPL {X  -162.820, Y  +601.090, Z    +0.000, E1   -58.519, E3 +262932.117}
SPL {X  -162.820, Y  +609.492, Z    +0.000, E1   -58.431, E3 +262943.422}
SPL {X  -162.820, Y  +617.241, Z    +0.000, E1   -58.340, E3 +262953.947}
SPL {X  -162.820, Y  +626.506, Z    +0.000, E1   -58.420, E3 +262965.329}
SPL {X  -162.820, Y  +638.850, Z    +0.000, E1   -58.527, E3 +262980.545}
SPL {X  -162.820, Y  +651.112, Z    +0.000, E1   -58.411, E3 +262996.903}
SPL {X  -162.820, Y  +660.924, Z    +0.000, E1   -58.393, E3 +263009.503}
SPL {X  -162.820, Y  +670.459, Z    +0.000, E1   -58.489, E3 +263021.104}
SPL {X  -162.713, Y  +679.396, Z    +0.000, E1   -58.414, E3 +263033.003}
SPL {X  -162.301, Y  +686.495, Z    +0.000, E1   -58.302, E3 +263042.787}
SPL {X  -161.571, Y  +693.631, Z    +0.000, E1   -58.186, E3 +263052.751}
SPL {X  -160.411, Y  +701.402, Z    +0.000, E1   -58.100, E3 +263063.227}
SPL {X  -159.229, Y  +707.508, Z    +0.000, E1   -57.870, E3 +263072.465}
SPL {X  -157.825, Y  +713.519, Z    +0.000, E1   -57.630, E3 +263081.701}
SPL {X  -156.079, Y  +719.864, Z    +0.000, E1   -57.324, E3 +263091.664}
SPL {X  -154.064, Y  +726.175, Z    +0.000, E1   -57.042, E3 +263101.426}
SPL {X  -152.053, Y  +731.726, Z    +0.000, E1   -56.648, E3 +263110.711}
SPL {X  -150.108, Y  +736.570, Z    +0.000, E1   -56.283, E3 +263118.950}
SPL {X  -147.726, Y  +741.964, Z    +0.000, E1   -55.884, E3 +263127.986}
SPL {X  -145.163, Y  +747.242, Z    +0.000, E1   -55.517, E3 +263136.582}
SPL {X  -142.489, Y  +752.286, Z    +0.000, E1   -55.227, E3 +263144.409}
SPL {X  -136.074, Y  +762.910, Z    +0.000, E1   -57.336, E3 +263147.531}
SPL {X  -116.561, Y  +787.183, Z    +0.000, E1   -51.088, E3 +263231.999}
ENDSPLINE

SPLINE
SPL {X  -119.623, Y  +783.957, Z    +0.000, E1   -49.202, E3 +263356.532}
SPL {X  -149.958, Y  +736.927, Z    +0.000, E1   -34.772, E3 +263354.249}
SPL {X  -158.826, Y  +709.343, Z    +0.000, E1   -23.029, E3 +263362.592}
SPL {X  -161.344, Y  +695.370, Z    +0.000, E1   -15.607, E3 +263364.991}
SPL {X  -162.477, Y  +684.065, Z    +0.000, E1    -8.887, E3 +263364.621}
SPL {X  -162.776, Y  +677.290, Z    +0.000, E1    -4.406, E3 +263365.293}
SPL {X  -162.820, Y  +673.886, Z    +0.000, E1    -1.998, E3 +263365.121}
SPL {X  -162.820, Y  +670.901, Z    +0.000, E1    +0.338, E3 +263364.555}
SPL {X  -162.820, Y  +667.984, Z    +0.000, E1    +3.594, E3 +263364.387}
SPL {X  -162.820, Y  +664.667, Z    +0.000, E1    +7.867, E3 +263364.100}
SPL {X  -162.820, Y  +660.022, Z    +0.000, E1   +14.535, E3 +263363.997}
SPL {X  -162.820, Y  +653.408, Z    +0.000, E1   +24.221, E3 +263364.307}
SPL {X  -162.820, Y  +640.244, Z    +0.000, E1   +41.042, E3 +263364.351}
SPL {X  -162.820, Y  +592.517, Z    +0.000, E1   +60.575, E3 +263383.482}
SPL {X  -162.820, Y  +515.613, Z    +0.000, E1   +60.751, E3 +263457.317}
ENDSPLINE

SPLINE
SPL {X  -162.820, Y  +518.198, Z    +0.000, E1   +58.338, E3 +263470.473}
ENDSPLINE

SPLINE
SPL {X  -162.820, Y  +508.314, Z    +0.000, E1   +58.337, E3 +263483.169}
SPL {X  -162.820, Y  +498.518, Z    +0.000, E1   +58.346, E3 +263495.675}
SPL {X  -162.820, Y  +489.418, Z    +0.000, E1   +58.357, E3 +263507.265}
SPL {X  -162.820, Y  +479.904, Z    +0.000, E1   +58.389, E3 +263519.312}
SPL {X  -162.820, Y  +472.095, Z    +0.000, E1   +58.202, E3 +263530.492}
SPL {X  -162.820, Y  +463.661, Z    +0.000, E1   +58.370, E3 +263540.278}
SPL {X  -162.820, Y  +454.904, Z    +0.000, E1   +58.380, E3 +263551.444}
SPL {X  -162.820, Y  +446.206, Z    +0.000, E1   +58.278, E3 +263563.335}
SPL {X  -162.820, Y  +436.416, Z    +0.000, E1   +58.325, E3 +263575.575}
SPL {X  -162.820, Y  +426.628, Z    +0.000, E1   +58.432, E3 +263587.443}
SPL {X  -162.820, Y  +415.377, Z    +0.000, E1   +58.239, E3 +263603.375}
SPL {X  -162.820, Y  +403.663, Z    +0.000, E1   +58.258, E3 +263618.154}
SPL {X  -162.820, Y  +397.157, Z    +0.000, E1   +58.054, E3 +263627.890}
SPL {X  -162.820, Y  +387.359, Z    +0.000, E1   +58.365, E3 +263638.519}
SPL {X  -162.810, Y  +378.731, Z    +0.000, E1   +58.366, E3 +263649.577}
SPL {X  -162.546, Y  +371.051, Z    +0.000, E1   +58.239, E3 +263660.297}
SPL {X  -161.863, Y  +362.875, Z    +0.000, E1   +58.273, E3 +263670.522}
SPL {X  -161.159, Y  +357.301, Z    +0.000, E1   +57.946, E3 +263679.822}
SPL {X  -159.864, Y  +349.614, Z    +0.000, E1   +57.922, E3 +263689.898}
SPL {X  -158.300, Y  +342.404, Z    +0.000, E1   +57.579, E3 +263701.344}
SPL {X  -156.187, Y  +334.499, Z    +0.000, E1   +57.331, E3 +263713.004}
SPL {X  -154.237, Y  +328.333, Z    +0.000, E1   +56.930, E3 +263723.214}
SPL {X  -152.732, Y  +324.078, Z    +0.000, E1   +56.482, E3 +263731.219}
SPL {X  -150.609, Y  +318.634, Z    +0.000, E1   +56.366, E3 +263738.913}
SPL {X  -148.206, Y  +313.080, Z    +0.000, E1   +55.888, E3 +263748.625}
SPL {X  -145.956, Y  +308.339, Z    +0.000, E1   +55.380, E3 +263757.301}
SPL {X  -143.330, Y  +303.254, Z    +0.000, E1   +55.057, E3 +263765.421}
SPL {X  -137.431, Y  +293.190, Z    +0.000, E1   +56.809, E3 +263769.584}
SPL {X  -115.845, Y  +266.087, Z    +0.000, E1   +50.276, E3 +263868.442}
SPL {X  -114.083, Y  +264.330, Z    +0.000, E1   +49.123, E3 +263907.152}
ENDSPLINE

SPLINE
SPL {X  -149.622, Y  +316.285, Z    +0.000, E1   +35.036, E3 +263975.664}
SPL {X  -158.704, Y  +344.121, Z    +0.000, E1   +23.312, E3 +263985.537}
SPL {X  -162.109, Y  +365.304, Z    +0.000, E1   +11.761, E3 +263984.839}
SPL {X  -162.811, Y  +378.776, Z    +0.000, E1    +3.078, E3 +263985.083}
SPL {X  -162.820, Y  +383.454, Z    +0.000, E1    -0.619, E3 +263984.551}
SPL {X  -162.820, Y  +387.033, Z    +0.000, E1    -4.758, E3 +263984.255}
SPL {X  -162.820, Y  +390.967, Z    +0.000, E1    -9.918, E3 +263984.700}
SPL {X  -162.820, Y  +397.718, Z    +0.000, E1   -19.761, E3 +263984.074}
SPL {X  -162.820, Y  +405.058, Z    +0.000, E1   -29.962, E3 +263984.987}
SPL {X  -162.820, Y  +417.515, Z    +0.000, E1   -44.878, E3 +263984.149}
SPL {X  -162.820, Y  +462.065, Z    +0.000, E1   -61.507, E3 +264001.109}
SPL {X  -162.820, Y  +504.602, Z    +0.000, E1   -64.286, E3 +264026.635}
SPL {X  -162.820, Y  +535.709, Z    +0.000, E1   -59.182, E3 +264084.314}
SPL {X  -162.820, Y  +543.678, Z    +0.000, E1   -58.515, E3 +264098.703}
SPL {X  -162.820, Y  +553.725, Z    +0.000, E1   -58.454, E3 +264111.964}
SPL {X  -162.820, Y  +562.850, Z    +0.000, E1   -58.373, E3 +264124.126}
SPL {X  -162.820, Y  +571.217, Z    +0.000, E1   -58.397, E3 +264134.679}
SPL {X  -162.820, Y  +581.879, Z    +0.000, E1   -58.475, E3 +264147.932}
SPL {X  -162.820, Y  +591.768, Z    +0.000, E1   -58.375, E3 +264161.130}
SPL {X  -162.820, Y  +601.090, Z    +0.000, E1   -58.519, E3 +264172.117}
SPL {X  -162.820, Y  +609.492, Z    +0.000, E1   -58.431, E3 +264183.422}
SPL {X  -162.820, Y  +617.241, Z    +0.000, E1   -58.340, E3 +264193.947}
SPL {X  -162.820, Y  +626.506, Z    +0.000, E1   -58.420, E3 +264205.329}
SPL {X  -162.820, Y  +638.850, Z    +0.000, E1   -58.527, E3 +264220.545}
SPL {X  -162.820, Y  +651.112, Z    +0.000, E1   -58.411, E3 +264236.903}
SPL {X  -162.820, Y  +660.924, Z    +0.000, E1   -58.393, E3 +264249.503}
SPL {X  -162.820, Y  +670.459, Z    +0.000, E1   -58.489, E3 +264261.104}
SPL {X  -162.713, Y  +679.396, Z    +0.000, E1   -58.414, E3 +264273.003}
SPL {X  -162.301, Y  +686.495, Z    +0.000, E1   -58.302, E3 +264282.787}
SPL {X  -161.571, Y  +693.631, Z    +0.000, E1   -58.186, E3 +264292.751}
SPL {X  -160.411, Y  +701.402, Z    +0.000, E1   -58.100, E3 +264303.227}
SPL {X  -159.229, Y  +707.508, Z    +0.000, E1   -57.870, E3 +264312.465}
SPL {X  -157.825, Y  +713.519, Z    +0.000, E1   -57.630, E3 +264321.701}
SPL {X  -156.079, Y  +719.864, Z    +0.000, E1   -57.324, E3 +264331.664}
SPL {X  -154.064, Y  +726.175, Z    +0.000, E1   -57.042, E3 +264341.426}
SPL {X  -152.053, Y  +731.726, Z    +0.000, E1   -56.648, E3 +264350.711}
SPL {X  -150.108, Y  +736.570, Z    +0.000, E1   -56.283, E3 +264358.950}
SPL {X  -147.726, Y  +741.964, Z    +0.000, E1   -55.884, E3 +264367.986}
SPL {X  -145.163, Y  +747.242, Z    +0.000, E1   -55.517, E3 +264376.582}
SPL {X  -142.489, Y  +752.286, Z    +0.000, E1   -55.227, E3 +264384.409}
SPL {X  -136.074, Y  +762.910, Z    +0.000, E1   -57.336, E3 +264387.531}
SPL {X  -116.561, Y  +787.183, Z    +0.000, E1   -51.088, E3 +264471.999}
ENDSPLINE

SPLINE
SPL {X  -119.623, Y  +783.957, Z    +0.000, E1   -49.202, E3 +264596.532}
SPL {X  -149.958, Y  +736.927, Z    +0.000, E1   -34.772, E3 +264594.249}
SPL {X  -158.826, Y  +709.343, Z    +0.000, E1   -23.029, E3 +264602.592}
SPL {X  -161.344, Y  +695.370, Z    +0.000, E1   -15.607, E3 +264604.991}
SPL {X  -162.477, Y  +684.065, Z    +0.000, E1    -8.887, E3 +264604.621}
SPL {X  -162.813, Y  +675.055, Z    +0.000, E1    -2.911, E3 +264605.184}
SPL {X  -162.820, Y  +670.901, Z    +0.000, E1    +0.338, E3 +264604.555}
SPL {X  -162.820, Y  +667.984, Z    +0.000, E1    +3.594, E3 +264604.387}
SPL {X  -162.820, Y  +664.667, Z    +0.000, E1    +7.867, E3 +264604.100}
SPL {X  -162.820, Y  +660.022, Z    +0.000, E1   +14.535, E3 +264603.997}
SPL {X  -162.820, Y  +653.408, Z    +0.000, E1   +24.221, E3 +264604.307}
SPL {X  -162.820, Y  +640.244, Z    +0.000, E1   +41.042, E3 +264604.351}
SPL {X  -162.820, Y  +592.517, Z    +0.000, E1   +60.575, E3 +264623.482}
SPL {X  -162.820, Y  +515.613, Z    +0.000, E1   +60.751, E3 +264697.317}
ENDSPLINE

SPLINE
SPL {X  -162.820, Y  +518.198, Z    +0.000, E1   +58.338, E3 +264710.473}
ENDSPLINE

SPLINE
SPL {X  -162.820, Y  +508.314, Z    +0.000, E1   +58.337, E3 +264723.169}
SPL {X  -162.820, Y  +498.518, Z    +0.000, E1   +58.346, E3 +264735.675}
SPL {X  -162.820, Y  +489.418, Z    +0.000, E1   +58.357, E3 +264747.265}
SPL {X  -162.820, Y  +479.904, Z    +0.000, E1   +58.389, E3 +264759.312}
SPL {X  -162.820, Y  +472.095, Z    +0.000, E1   +58.202, E3 +264770.492}
SPL {X  -162.820, Y  +463.661, Z    +0.000, E1   +58.370, E3 +264780.278}
SPL {X  -162.820, Y  +454.904, Z    +0.000, E1   +58.380, E3 +264791.444}
SPL {X  -162.820, Y  +446.206, Z    +0.000, E1   +58.278, E3 +264803.335}
SPL {X  -162.820, Y  +436.416, Z    +0.000, E1   +58.325, E3 +264815.575}
SPL {X  -162.820, Y  +426.628, Z    +0.000, E1   +58.432, E3 +264827.443}
SPL {X  -162.820, Y  +418.389, Z    +0.000, E1   +58.300, E3 +264838.846}
SPL {X  -162.820, Y  +412.292, Z    +0.000, E1   +58.070, E3 +264848.214}
SPL {X  -162.820, Y  +403.663, Z    +0.000, E1   +58.258, E3 +264858.154}
SPL {X  -162.820, Y  +397.157, Z    +0.000, E1   +58.054, E3 +264867.890}
SPL {X  -162.820, Y  +387.359, Z    +0.000, E1   +58.365, E3 +264878.519}
SPL {X  -162.810, Y  +378.731, Z    +0.000, E1   +58.366, E3 +264889.577}
SPL {X  -162.546, Y  +371.051, Z    +0.000, E1   +58.239, E3 +264900.297}
SPL {X  -161.863, Y  +362.875, Z    +0.000, E1   +58.273, E3 +264910.522}
SPL {X  -161.159, Y  +357.301, Z    +0.000, E1   +57.946, E3 +264919.822}
SPL {X  -159.864, Y  +349.614, Z    +0.000, E1   +57.922, E3 +264929.898}
SPL {X  -158.300, Y  +342.404, Z    +0.000, E1   +57.579, E3 +264941.344}
SPL {X  -156.187, Y  +334.499, Z    +0.000, E1   +57.331, E3 +264953.004}
SPL {X  -154.237, Y  +328.333, Z    +0.000, E1   +56.930, E3 +264963.214}
SPL {X  -152.732, Y  +324.078, Z    +0.000, E1   +56.482, E3 +264971.219}
SPL {X  -150.609, Y  +318.634, Z    +0.000, E1   +56.366, E3 +264978.913}
SPL {X  -148.206, Y  +313.080, Z    +0.000, E1   +55.888, E3 +264988.625}
SPL {X  -145.956, Y  +308.339, Z    +0.000, E1   +55.380, E3 +264997.301}
SPL {X  -143.330, Y  +303.254, Z    +0.000, E1   +55.057, E3 +265005.421}
SPL {X  -137.431, Y  +293.190, Z    +0.000, E1   +56.809, E3 +265009.584}
SPL {X  -115.845, Y  +266.087, Z    +0.000, E1   +50.276, E3 +265108.442}
SPL {X  -114.083, Y  +264.330, Z    +0.000, E1   +49.123, E3 +265147.152}
ENDSPLINE

SPLINE
SPL {X  -149.622, Y  +316.285, Z    +0.000, E1   +35.036, E3 +265215.664}
SPL {X  -158.704, Y  +344.121, Z    +0.000, E1   +23.312, E3 +265225.537}
SPL {X  -161.701, Y  +361.440, Z    +0.000, E1   +13.961, E3 +265224.608}
SPL {X  -162.691, Y  +374.019, Z    +0.000, E1    +6.263, E3 +265225.261}
SPL {X  -162.820, Y  +381.771, Z    +0.000, E1    +0.850, E3 +265224.745}
SPL {X  -162.820, Y  +384.317, Z    +0.000, E1    -1.618, E3 +265224.463}
SPL {X  -162.820, Y  +387.033, Z    +0.000, E1    -4.758, E3 +265224.255}
SPL {X  -162.820, Y  +390.967, Z    +0.000, E1    -9.918, E3 +265224.700}
SPL {X  -162.820, Y  +395.392, Z    +0.000, E1   -16.726, E3 +265223.141}
SPL {X  -162.820, Y  +402.654, Z    +0.000, E1   -26.492, E3 +265225.032}
SPL {X  -162.820, Y  +417.515, Z    +0.000, E1   -44.878, E3 +265224.149}
SPL {X  -162.820, Y  +462.065, Z    +0.000, E1   -61.507, E3 +265241.109}
SPL {X  -162.820, Y  +504.602, Z    +0.000, E1   -64.286, E3 +265266.635}
SPL {X  -162.820, Y  +539.530, Z    +0.000, E1   -60.821, E3 +265317.326}
ENDSPLINE

SPLINE
SPL {X  -162.820, Y  +534.172, Z    +0.000, E1   -58.470, E3 +265326.826}
ENDSPLINE

SPLINE
SPL {X  -162.820, Y  +543.678, Z    +0.000, E1   -58.515, E3 +265338.703}
SPL {X  -162.820, Y  +553.725, Z    +0.000, E1   -58.454, E3 +265351.964}
SPL {X  -162.820, Y  +562.850, Z    +0.000, E1   -58.373, E3 +265364.126}
SPL {X  -162.820, Y  +573.452, Z    +0.000, E1   -58.444, E3 +265377.339}
SPL {X  -162.820, Y  +583.632, Z    +0.000, E1   -58.444, E3 +265390.266}
SPL {X  -162.820, Y  +591.768, Z    +0.000, E1   -58.375, E3 +265401.130}
SPL {X  -162.820, Y  +601.090, Z    +0.000, E1   -58.519, E3 +265412.117}
SPL {X  -162.820, Y  +609.492, Z    +0.000, E1   -58.431, E3 +265423.422}
SPL {X  -162.820, Y  +617.241, Z    +0.000, E1   -58.340, E3 +265433.947}
SPL {X  -162.820, Y  +626.506, Z    +0.000, E1   -58.420, E3 +265445.329}
SPL {X  -162.820, Y  +635.919, Z    +0.000, E1   -58.604, E3 +265456.073}
SPL {X  -162.820, Y  +643.895, Z    +0.000, E1   -58.380, E3 +265467.838}
SPL {X  -162.820, Y  +653.118, Z    +0.000, E1   -58.401, E3 +265479.435}
SPL {X  -162.820, Y  +660.924, Z    +0.000, E1   -58.393, E3 +265489.503}
SPL {X  -162.820, Y  +670.459, Z    +0.000, E1   -58.489, E3 +265501.104}
SPL {X  -162.713, Y  +679.396, Z    +0.000, E1   -58.414, E3 +265513.003}
SPL {X  -162.301, Y  +686.495, Z    +0.000, E1   -58.302, E3 +265522.787}
SPL {X  -161.571, Y  +693.631, Z    +0.000, E1   -58.186, E3 +265532.751}
SPL {X  -160.411, Y  +701.402, Z    +0.000, E1   -58.100, E3 +265543.227}
SPL {X  -159.229, Y  +707.508, Z    +0.000, E1   -57.870, E3 +265552.465}
SPL {X  -157.825, Y  +713.519, Z    +0.000, E1   -57.630, E3 +265561.701}
SPL {X  -156.079, Y  +719.864, Z    +0.000, E1   -57.324, E3 +265571.664}
SPL {X  -154.064, Y  +726.175, Z    +0.000, E1   -57.042, E3 +265581.426}
SPL {X  -152.053, Y  +731.726, Z    +0.000, E1   -56.648, E3 +265590.711}
SPL {X  -150.108, Y  +736.570, Z    +0.000, E1   -56.283, E3 +265598.950}
SPL {X  -147.726, Y  +741.964, Z    +0.000, E1   -55.884, E3 +265607.986}
SPL {X  -145.163, Y  +747.242, Z    +0.000, E1   -55.517, E3 +265616.582}
SPL {X  -142.489, Y  +752.286, Z    +0.000, E1   -55.227, E3 +265624.409}
SPL {X  -136.074, Y  +762.910, Z    +0.000, E1   -57.336, E3 +265627.531}
SPL {X  -116.561, Y  +787.183, Z    +0.000, E1   -51.088, E3 +265711.999}
ENDSPLINE

SPLINE
SPL {X  -119.623, Y  +783.957, Z    +0.000, E1   -49.202, E3 +265836.532}
SPL {X  -149.958, Y  +736.927, Z    +0.000, E1   -34.772, E3 +265834.249}
SPL {X  -158.826, Y  +709.343, Z    +0.000, E1   -23.029, E3 +265842.592}
SPL {X  -161.344, Y  +695.370, Z    +0.000, E1   -15.607, E3 +265844.991}
SPL {X  -162.477, Y  +684.065, Z    +0.000, E1    -8.887, E3 +265844.621}
SPL {X  -162.813, Y  +675.055, Z    +0.000, E1    -2.911, E3 +265845.184}
SPL {X  -162.820, Y  +670.901, Z    +0.000, E1    +0.338, E3 +265844.555}
SPL {X  -162.820, Y  +667.984, Z    +0.000, E1    +3.594, E3 +265844.387}
SPL {X  -162.820, Y  +664.667, Z    +0.000, E1    +7.867, E3 +265844.100}
SPL {X  -162.820, Y  +660.022, Z    +0.000, E1   +14.535, E3 +265843.997}
SPL {X  -162.820, Y  +653.408, Z    +0.000, E1   +24.221, E3 +265844.307}
SPL {X  -162.820, Y  +640.244, Z    +0.000, E1   +41.042, E3 +265844.351}
SPL {X  -162.820, Y  +592.517, Z    +0.000, E1   +60.575, E3 +265863.482}
SPL {X  -162.820, Y  +515.613, Z    +0.000, E1   +60.751, E3 +265937.317}
ENDSPLINE

SPLINE
SPL {X  -162.820, Y  +518.198, Z    +0.000, E1   +58.338, E3 +265950.473}
ENDSPLINE

SPLINE
SPL {X  -162.820, Y  +508.314, Z    +0.000, E1   +58.337, E3 +265963.169}
SPL {X  -162.820, Y  +498.518, Z    +0.000, E1   +58.346, E3 +265975.675}
SPL {X  -162.820, Y  +489.418, Z    +0.000, E1   +58.357, E3 +265987.265}
SPL {X  -162.820, Y  +479.904, Z    +0.000, E1   +58.389, E3 +265999.312}
SPL {X  -162.820, Y  +472.095, Z    +0.000, E1   +58.202, E3 +266010.492}
SPL {X  -162.820, Y  +463.661, Z    +0.000, E1   +58.370, E3 +266020.278}
SPL {X  -162.820, Y  +454.904, Z    +0.000, E1   +58.380, E3 +266031.444}
SPL {X  -162.820, Y  +446.206, Z    +0.000, E1   +58.278, E3 +266043.335}
SPL {X  -162.820, Y  +436.416, Z    +0.000, E1   +58.325, E3 +266055.575}
SPL {X  -162.820, Y  +426.628, Z    +0.000, E1   +58.432, E3 +266067.443}
SPL {X  -162.820, Y  +415.377, Z    +0.000, E1   +58.239, E3 +266083.375}
SPL {X  -162.820, Y  +403.663, Z    +0.000, E1   +58.258, E3 +266098.154}
SPL {X  -162.820, Y  +397.157, Z    +0.000, E1   +58.054, E3 +266107.890}
SPL {X  -162.820, Y  +387.359, Z    +0.000, E1   +58.365, E3 +266118.519}
SPL {X  -162.810, Y  +378.731, Z    +0.000, E1   +58.366, E3 +266129.577}
SPL {X  -162.546, Y  +371.051, Z    +0.000, E1   +58.239, E3 +266140.297}
SPL {X  -161.863, Y  +362.875, Z    +0.000, E1   +58.273, E3 +266150.522}
SPL {X  -161.159, Y  +357.301, Z    +0.000, E1   +57.946, E3 +266159.822}
SPL {X  -159.864, Y  +349.614, Z    +0.000, E1   +57.922, E3 +266169.898}
SPL {X  -158.548, Y  +343.449, Z    +0.000, E1   +57.711, E3 +266179.072}
SPL {X  -156.580, Y  +335.856, Z    +0.000, E1   +57.340, E3 +266191.295}
SPL {X  -154.237, Y  +328.333, Z    +0.000, E1   +56.930, E3 +266203.214}
SPL {X  -152.732, Y  +324.078, Z    +0.000, E1   +56.482, E3 +266211.219}
SPL {X  -150.609, Y  +318.634, Z    +0.000, E1   +56.366, E3 +266218.913}
SPL {X  -148.206, Y  +313.080, Z    +0.000, E1   +55.888, E3 +266228.625}
SPL {X  -145.956, Y  +308.339, Z    +0.000, E1   +55.380, E3 +266237.301}
SPL {X  -143.330, Y  +303.254, Z    +0.000, E1   +55.057, E3 +266245.421}
SPL {X  -137.431, Y  +293.190, Z    +0.000, E1   +56.809, E3 +266249.584}
SPL {X  -115.845, Y  +266.087, Z    +0.000, E1   +50.276, E3 +266348.442}
SPL {X  -114.083, Y  +264.330, Z    +0.000, E1   +49.123, E3 +266387.152}
ENDSPLINE

SPLINE
SPL {X  -149.622, Y  +316.285, Z    +0.000, E1   +35.036, E3 +266455.664}
SPL {X  -158.704, Y  +344.121, Z    +0.000, E1   +23.312, E3 +266465.537}
SPL {X  -162.109, Y  +365.304, Z    +0.000, E1   +11.761, E3 +266464.839}
SPL {X  -162.811, Y  +378.776, Z    +0.000, E1    +3.078, E3 +266465.083}
SPL {X  -162.820, Y  +383.454, Z    +0.000, E1    -0.619, E3 +266464.551}
SPL {X  -162.820, Y  +387.033, Z    +0.000, E1    -4.758, E3 +266464.255}
SPL {X  -162.820, Y  +390.967, Z    +0.000, E1    -9.918, E3 +266464.700}
SPL {X  -162.820, Y  +397.718, Z    +0.000, E1   -19.761, E3 +266464.074}
SPL {X  -162.820, Y  +405.058, Z    +0.000, E1   -29.962, E3 +266464.987}
SPL {X  -162.820, Y  +417.515, Z    +0.000, E1   -44.878, E3 +266464.149}
SPL {X  -162.820, Y  +462.065, Z    +0.000, E1   -61.507, E3 +266481.109}
SPL {X  -162.820, Y  +504.602, Z    +0.000, E1   -64.286, E3 +266506.635}
SPL {X  -162.820, Y  +539.530, Z    +0.000, E1   -60.821, E3 +266557.326}
ENDSPLINE

SPLINE
SPL {X  -162.820, Y  +534.172, Z    +0.000, E1   -58.470, E3 +266566.826}
ENDSPLINE

SPLINE
SPL {X  -162.820, Y  +543.678, Z    +0.000, E1   -58.515, E3 +266578.703}
SPL {X  -162.820, Y  +553.725, Z    +0.000, E1   -58.454, E3 +266591.964}
SPL {X  -162.820, Y  +562.850, Z    +0.000, E1   -58.373, E3 +266604.126}
SPL {X  -162.820, Y  +573.452, Z    +0.000, E1   -58.444, E3 +266617.339}
SPL {X  -162.820, Y  +583.632, Z    +0.000, E1   -58.444, E3 +266630.266}
SPL {X  -162.820, Y  +591.768, Z    +0.000, E1   -58.375, E3 +266641.130}
SPL {X  -162.820, Y  +601.090, Z    +0.000, E1   -58.519, E3 +266652.117}
SPL {X  -162.820, Y  +609.492, Z    +0.000, E1   -58.431, E3 +266663.422}
SPL {X  -162.820, Y  +617.241, Z    +0.000, E1   -58.340, E3 +266673.947}
SPL {X  -162.820, Y  +626.506, Z    +0.000, E1   -58.420, E3 +266685.329}
SPL {X  -162.820, Y  +635.919, Z    +0.000, E1   -58.604, E3 +266696.073}
SPL {X  -162.820, Y  +643.895, Z    +0.000, E1   -58.380, E3 +266707.838}
SPL {X  -162.820, Y  +653.118, Z    +0.000, E1   -58.401, E3 +266719.435}
SPL {X  -162.820, Y  +660.924, Z    +0.000, E1   -58.393, E3 +266729.503}
SPL {X  -162.820, Y  +670.459, Z    +0.000, E1   -58.489, E3 +266741.104}
SPL {X  -162.713, Y  +679.396, Z    +0.000, E1   -58.414, E3 +266753.003}
SPL {X  -162.301, Y  +686.495, Z    +0.000, E1   -58.302, E3 +266762.787}
SPL {X  -161.571, Y  +693.631, Z    +0.000, E1   -58.186, E3 +266772.751}
SPL {X  -160.411, Y  +701.402, Z    +0.000, E1   -58.100, E3 +266783.227}
SPL {X  -159.229, Y  +707.508, Z    +0.000, E1   -57.870, E3 +266792.465}
SPL {X  -157.825, Y  +713.519, Z    +0.000, E1   -57.630, E3 +266801.701}
SPL {X  -156.079, Y  +719.864, Z    +0.000, E1   -57.324, E3 +266811.664}
SPL {X  -154.064, Y  +726.175, Z    +0.000, E1   -57.042, E3 +266821.426}
SPL {X  -152.053, Y  +731.726, Z    +0.000, E1   -56.648, E3 +266830.711}
SPL {X  -150.108, Y  +736.570, Z    +0.000, E1   -56.283, E3 +266838.950}
SPL {X  -147.726, Y  +741.964, Z    +0.000, E1   -55.884, E3 +266847.986}
SPL {X  -145.163, Y  +747.242, Z    +0.000, E1   -55.517, E3 +266856.582}
SPL {X  -142.489, Y  +752.286, Z    +0.000, E1   -55.227, E3 +266864.409}
SPL {X  -136.074, Y  +762.910, Z    +0.000, E1   -57.336, E3 +266867.531}
SPL {X  -116.561, Y  +787.183, Z    +0.000, E1   -51.088, E3 +266951.999}
ENDSPLINE

SPLINE
SPL {X  -119.623, Y  +783.957, Z    +0.000, E1   -49.202, E3 +267076.532}
SPL {X  -149.958, Y  +736.927, Z    +0.000, E1   -34.772, E3 +267074.249}
SPL {X  -158.826, Y  +709.343, Z    +0.000, E1   -23.029, E3 +267082.592}
SPL {X  -161.800, Y  +691.694, Z    +0.000, E1   -13.520, E3 +267084.886}
SPL {X  -162.711, Y  +679.444, Z    +0.000, E1    -5.922, E3 +267084.960}
SPL {X  -162.820, Y  +672.303, Z    +0.000, E1    -0.875, E3 +267084.825}
SPL {X  -162.820, Y  +669.030, Z    +0.000, E1    +2.242, E3 +267084.397}
SPL {X  -162.820, Y  +664.667, Z    +0.000, E1    +7.867, E3 +267084.100}
SPL {X  -162.820, Y  +660.022, Z    +0.000, E1   +14.535, E3 +267083.997}
SPL {X  -162.820, Y  +653.408, Z    +0.000, E1   +24.221, E3 +267084.307}
SPL {X  -162.820, Y  +640.244, Z    +0.000, E1   +41.042, E3 +267084.351}
SPL {X  -162.820, Y  +592.517, Z    +0.000, E1   +60.575, E3 +267103.482}
SPL {X  -162.820, Y  +515.613, Z    +0.000, E1   +60.751, E3 +267177.317}
ENDSPLINE

SPLINE
SPL {X  -162.820, Y  +518.198, Z    +0.000, E1   +58.338, E3 +267190.473}
ENDSPLINE

SPLINE
SPL {X  -162.820, Y  +508.314, Z    +0.000, E1   +58.337, E3 +267203.169}
SPL {X  -162.820, Y  +498.518, Z    +0.000, E1   +58.346, E3 +267215.675}
SPL {X  -162.820, Y  +489.418, Z    +0.000, E1   +58.357, E3 +267227.265}
SPL {X  -162.820, Y  +479.904, Z    +0.000, E1   +58.389, E3 +267239.312}
SPL {X  -162.820, Y  +472.095, Z    +0.000, E1   +58.202, E3 +267250.492}
SPL {X  -162.820, Y  +463.661, Z    +0.000, E1   +58.370, E3 +267260.278}
SPL {X  -162.820, Y  +454.904, Z    +0.000, E1   +58.380, E3 +267271.444}
SPL {X  -162.820, Y  +446.206, Z    +0.000, E1   +58.278, E3 +267283.335}
SPL {X  -162.820, Y  +436.416, Z    +0.000, E1   +58.325, E3 +267295.575}
SPL {X  -162.820, Y  +426.628, Z    +0.000, E1   +58.432, E3 +267307.443}
SPL {X  -162.820, Y  +415.377, Z    +0.000, E1   +58.239, E3 +267323.375}
SPL {X  -162.820, Y  +403.663, Z    +0.000, E1   +58.258, E3 +267338.154}
SPL {X  -162.820, Y  +397.157, Z    +0.000, E1   +58.054, E3 +267347.890}
SPL {X  -162.820, Y  +387.359, Z    +0.000, E1   +58.365, E3 +267358.519}
SPL {X  -162.810, Y  +378.731, Z    +0.000, E1   +58.366, E3 +267369.577}
SPL {X  -162.546, Y  +371.051, Z    +0.000, E1   +58.239, E3 +267380.297}
SPL {X  -161.863, Y  +362.875, Z    +0.000, E1   +58.273, E3 +267390.522}
SPL {X  -161.159, Y  +357.301, Z    +0.000, E1   +57.946, E3 +267399.822}
SPL {X  -159.864, Y  +349.614, Z    +0.000, E1   +57.922, E3 +267409.898}
SPL {X  -158.548, Y  +343.449, Z    +0.000, E1   +57.711, E3 +267419.072}
SPL {X  -156.580, Y  +335.856, Z    +0.000, E1   +57.340, E3 +267431.295}
SPL {X  -154.237, Y  +328.333, Z    +0.000, E1   +56.930, E3 +267443.214}
SPL {X  -152.732, Y  +324.078, Z    +0.000, E1   +56.482, E3 +267451.219}
SPL {X  -150.609, Y  +318.634, Z    +0.000, E1   +56.366, E3 +267458.913}
SPL {X  -148.206, Y  +313.080, Z    +0.000, E1   +55.888, E3 +267468.625}
SPL {X  -145.956, Y  +308.339, Z    +0.000, E1   +55.380, E3 +267477.301}
SPL {X  -142.234, Y  +301.255, Z    +0.000, E1   +55.418, E3 +267486.175}
SPL {X  -134.491, Y  +288.726, Z    +0.000, E1   +57.448, E3 +267491.831}
SPL {X  -115.845, Y  +266.087, Z    +0.000, E1   +50.276, E3 +267588.442}
SPL {X  -114.083, Y  +264.330, Z    +0.000, E1   +49.123, E3 +267627.152}
ENDSPLINE

SPLINE
SPL {X  -136.188, Y  +291.263, Z    +0.000, E1   +45.457, E3 +267723.218}
SPL {X  -151.738, Y  +321.457, Z    +0.000, E1   +32.773, E3 +267690.387}
SPL {X  -158.704, Y  +344.121, Z    +0.000, E1   +23.312, E3 +267705.537}
SPL {X  -162.109, Y  +365.304, Z    +0.000, E1   +11.761, E3 +267704.839}
SPL {X  -162.811, Y  +378.776, Z    +0.000, E1    +3.078, E3 +267705.083}
SPL {X  -162.820, Y  +382.545, Z    +0.000, E1    +0.100, E3 +267704.644}
SPL {X  -162.820, Y  +384.317, Z    +0.000, E1    -1.618, E3 +267704.463}
SPL {X  -162.820, Y  +387.033, Z    +0.000, E1    -4.758, E3 +267704.255}
SPL {X  -162.820, Y  +390.967, Z    +0.000, E1    -9.918, E3 +267704.700}
SPL {X  -162.820, Y  +395.392, Z    +0.000, E1   -16.726, E3 +267703.141}
SPL {X  -162.820, Y  +402.654, Z    +0.000, E1   -26.492, E3 +267705.032}
SPL {X  -162.820, Y  +417.515, Z    +0.000, E1   -44.878, E3 +267704.149}
SPL {X  -162.820, Y  +462.065, Z    +0.000, E1   -61.507, E3 +267721.109}
SPL {X  -162.820, Y  +504.602, Z    +0.000, E1   -64.286, E3 +267746.635}
SPL {X  -162.820, Y  +535.709, Z    +0.000, E1   -59.182, E3 +267804.314}
SPL {X  -162.820, Y  +543.678, Z    +0.000, E1   -58.515, E3 +267818.703}
SPL {X  -162.820, Y  +553.725, Z    +0.000, E1   -58.454, E3 +267831.964}
SPL {X  -162.820, Y  +562.850, Z    +0.000, E1   -58.373, E3 +267844.126}
SPL {X  -162.820, Y  +573.452, Z    +0.000, E1   -58.444, E3 +267857.339}
SPL {X  -162.820, Y  +583.632, Z    +0.000, E1   -58.444, E3 +267870.266}
SPL {X  -162.820, Y  +591.768, Z    +0.000, E1   -58.375, E3 +267881.130}
SPL {X  -162.820, Y  +601.090, Z    +0.000, E1   -58.519, E3 +267892.117}
SPL {X  -162.820, Y  +609.492, Z    +0.000, E1   -58.431, E3 +267903.422}
SPL {X  -162.820, Y  +617.241, Z    +0.000, E1   -58.340, E3 +267913.947}
SPL {X  -162.820, Y  +626.506, Z    +0.000, E1   -58.420, E3 +267925.329}
SPL {X  -162.820, Y  +638.850, Z    +0.000, E1   -58.527, E3 +267940.545}
SPL {X  -162.820, Y  +651.112, Z    +0.000, E1   -58.411, E3 +267956.903}
SPL {X  -162.820, Y  +660.924, Z    +0.000, E1   -58.393, E3 +267969.503}
SPL {X  -162.820, Y  +670.459, Z    +0.000, E1   -58.489, E3 +267981.104}
SPL {X  -162.713, Y  +679.396, Z    +0.000, E1   -58.414, E3 +267993.003}
SPL {X  -162.301, Y  +686.495, Z    +0.000, E1   -58.302, E3 +268002.787}
SPL {X  -161.571, Y  +693.631, Z    +0.000, E1   -58.186, E3 +268012.751}
SPL {X  -160.411, Y  +701.402, Z    +0.000, E1   -58.100, E3 +268023.227}
SPL {X  -159.229, Y  +707.508, Z    +0.000, E1   -57.870, E3 +268032.465}
SPL {X  -157.825, Y  +713.519, Z    +0.000, E1   -57.630, E3 +268041.701}
SPL {X  -156.079, Y  +719.864, Z    +0.000, E1   -57.324, E3 +268051.664}
SPL {X  -154.064, Y  +726.175, Z    +0.000, E1   -57.042, E3 +268061.426}
SPL {X  -152.053, Y  +731.726, Z    +0.000, E1   -56.648, E3 +268070.711}
SPL {X  -150.108, Y  +736.570, Z    +0.000, E1   -56.283, E3 +268078.950}
SPL {X  -147.726, Y  +741.964, Z    +0.000, E1   -55.884, E3 +268087.986}
SPL {X  -145.163, Y  +747.242, Z    +0.000, E1   -55.517, E3 +268096.582}
SPL {X  -142.489, Y  +752.286, Z    +0.000, E1   -55.227, E3 +268104.409}
SPL {X  -136.074, Y  +762.910, Z    +0.000, E1   -57.336, E3 +268107.531}
SPL {X  -116.561, Y  +787.183, Z    +0.000, E1   -51.088, E3 +268191.999}
ENDSPLINE

SPLINE
SPL {X  -119.623, Y  +783.957, Z    +0.000, E1   -49.202, E3 +268316.532}
SPL {X  -149.958, Y  +736.927, Z    +0.000, E1   -34.772, E3 +268314.249}
SPL {X  -158.826, Y  +709.343, Z    +0.000, E1   -23.029, E3 +268322.592}
SPL {X  -161.344, Y  +695.370, Z    +0.000, E1   -15.607, E3 +268324.991}
SPL {X  -162.477, Y  +684.065, Z    +0.000, E1    -8.887, E3 +268324.621}
SPL {X  -162.776, Y  +677.290, Z    +0.000, E1    -4.406, E3 +268325.293}
SPL {X  -162.820, Y  +673.886, Z    +0.000, E1    -1.998, E3 +268325.121}
SPL {X  -162.820, Y  +670.901, Z    +0.000, E1    +0.338, E3 +268324.555}
SPL {X  -162.820, Y  +667.984, Z    +0.000, E1    +3.594, E3 +268324.387}
SPL {X  -162.820, Y  +664.667, Z    +0.000, E1    +7.867, E3 +268324.100}
SPL {X  -162.820, Y  +660.022, Z    +0.000, E1   +14.535, E3 +268323.997}
SPL {X  -162.820, Y  +653.408, Z    +0.000, E1   +24.221, E3 +268324.307}
SPL {X  -162.820, Y  +640.244, Z    +0.000, E1   +41.042, E3 +268324.351}
SPL {X  -162.820, Y  +592.517, Z    +0.000, E1   +60.575, E3 +268343.482}
SPL {X  -162.820, Y  +515.613, Z    +0.000, E1   +60.751, E3 +268417.317}
ENDSPLINE

SPLINE
SPL {X  -162.820, Y  +518.198, Z    +0.000, E1   +58.338, E3 +268430.473}
ENDSPLINE

SPLINE
SPL {X  -162.820, Y  +508.314, Z    +0.000, E1   +58.337, E3 +268443.169}
SPL {X  -162.820, Y  +498.518, Z    +0.000, E1   +58.346, E3 +268455.675}
SPL {X  -162.820, Y  +489.418, Z    +0.000, E1   +58.357, E3 +268467.265}
SPL {X  -162.820, Y  +479.904, Z    +0.000, E1   +58.389, E3 +268479.312}
SPL {X  -162.820, Y  +472.095, Z    +0.000, E1   +58.202, E3 +268490.492}
SPL {X  -162.820, Y  +463.661, Z    +0.000, E1   +58.370, E3 +268500.278}
SPL {X  -162.820, Y  +454.904, Z    +0.000, E1   +58.380, E3 +268511.444}
SPL {X  -162.820, Y  +446.206, Z    +0.000, E1   +58.278, E3 +268523.335}
SPL {X  -162.820, Y  +436.416, Z    +0.000, E1   +58.325, E3 +268535.575}
SPL {X  -162.820, Y  +426.628, Z    +0.000, E1   +58.432, E3 +268547.443}
SPL {X  -162.820, Y  +415.377, Z    +0.000, E1   +58.239, E3 +268563.375}
SPL {X  -162.820, Y  +403.663, Z    +0.000, E1   +58.258, E3 +268578.154}
SPL {X  -162.820, Y  +397.157, Z    +0.000, E1   +58.054, E3 +268587.890}
SPL {X  -162.820, Y  +387.359, Z    +0.000, E1   +58.365, E3 +268598.519}
SPL {X  -162.810, Y  +378.731, Z    +0.000, E1   +58.366, E3 +268609.577}
SPL {X  -162.546, Y  +371.051, Z    +0.000, E1   +58.239, E3 +268620.297}
SPL {X  -161.863, Y  +362.875, Z    +0.000, E1   +58.273, E3 +268630.522}
SPL {X  -161.159, Y  +357.301, Z    +0.000, E1   +57.946, E3 +268639.822}
SPL {X  -159.864, Y  +349.614, Z    +0.000, E1   +57.922, E3 +268649.898}
SPL {X  -158.300, Y  +342.404, Z    +0.000, E1   +57.579, E3 +268661.344}
SPL {X  -156.187, Y  +334.499, Z    +0.000, E1   +57.331, E3 +268673.004}
SPL {X  -154.237, Y  +328.333, Z    +0.000, E1   +56.930, E3 +268683.214}
SPL {X  -152.732, Y  +324.078, Z    +0.000, E1   +56.482, E3 +268691.219}
SPL {X  -150.609, Y  +318.634, Z    +0.000, E1   +56.366, E3 +268698.913}
SPL {X  -148.206, Y  +313.080, Z    +0.000, E1   +55.888, E3 +268708.625}
SPL {X  -145.956, Y  +308.339, Z    +0.000, E1   +55.380, E3 +268717.301}
SPL {X  -143.330, Y  +303.254, Z    +0.000, E1   +55.057, E3 +268725.421}
SPL {X  -137.431, Y  +293.190, Z    +0.000, E1   +56.809, E3 +268729.584}
SPL {X  -115.845, Y  +266.087, Z    +0.000, E1   +50.276, E3 +268828.442}
SPL {X  -114.083, Y  +264.330, Z    +0.000, E1   +49.123, E3 +268867.152}
ENDSPLINE

SPLINE
SPL {X  -149.622, Y  +316.285, Z    +0.000, E1   +35.036, E3 +268935.664}
SPL {X  -158.704, Y  +344.121, Z    +0.000, E1   +23.312, E3 +268945.537}
SPL {X  -162.109, Y  +365.304, Z    +0.000, E1   +11.761, E3 +268944.839}
SPL {X  -162.811, Y  +378.776, Z    +0.000, E1    +3.078, E3 +268945.083}
SPL {X  -162.820, Y  +383.454, Z    +0.000, E1    -0.619, E3 +268944.551}
SPL {X  -162.820, Y  +387.033, Z    +0.000, E1    -4.758, E3 +268944.255}
SPL {X  -162.820, Y  +390.967, Z    +0.000, E1    -9.918, E3 +268944.700}
SPL {X  -162.820, Y  +397.718, Z    +0.000, E1   -19.761, E3 +268944.074}
SPL {X  -162.820, Y  +405.058, Z    +0.000, E1   -29.962, E3 +268944.987}
SPL {X  -162.820, Y  +417.515, Z    +0.000, E1   -44.878, E3 +268944.149}
SPL {X  -162.820, Y  +462.065, Z    +0.000, E1   -61.507, E3 +268961.109}
SPL {X  -162.820, Y  +504.602, Z    +0.000, E1   -64.286, E3 +268986.635}
SPL {X  -162.820, Y  +535.709, Z    +0.000, E1   -59.182, E3 +269044.314}
SPL {X  -162.820, Y  +543.678, Z    +0.000, E1   -58.515, E3 +269058.703}
SPL {X  -162.820, Y  +553.725, Z    +0.000, E1   -58.454, E3 +269071.964}
SPL {X  -162.820, Y  +562.850, Z    +0.000, E1   -58.373, E3 +269084.126}
SPL {X  -162.820, Y  +571.217, Z    +0.000, E1   -58.397, E3 +269094.679}
SPL {X  -162.820, Y  +581.879, Z    +0.000, E1   -58.475, E3 +269107.932}
SPL {X  -162.820, Y  +591.768, Z    +0.000, E1   -58.375, E3 +269121.130}
SPL {X  -162.820, Y  +601.090, Z    +0.000, E1   -58.519, E3 +269132.117}
SPL {X  -162.820, Y  +609.492, Z    +0.000, E1   -58.431, E3 +269143.422}
SPL {X  -162.820, Y  +617.241, Z    +0.000, E1   -58.340, E3 +269153.947}
SPL {X  -162.820, Y  +626.506, Z    +0.000, E1   -58.420, E3 +269165.329}
SPL {X  -162.820, Y  +638.850, Z    +0.000, E1   -58.527, E3 +269180.545}
SPL {X  -162.820, Y  +651.112, Z    +0.000, E1   -58.411, E3 +269196.903}
SPL {X  -162.820, Y  +660.924, Z    +0.000, E1   -58.393, E3 +269209.503}
SPL {X  -162.820, Y  +670.459, Z    +0.000, E1   -58.489, E3 +269221.104}
SPL {X  -162.713, Y  +679.396, Z    +0.000, E1   -58.414, E3 +269233.003}
SPL {X  -162.301, Y  +686.495, Z    +0.000, E1   -58.302, E3 +269242.787}
SPL {X  -161.571, Y  +693.631, Z    +0.000, E1   -58.186, E3 +269252.751}
SPL {X  -160.411, Y  +701.402, Z    +0.000, E1   -58.100, E3 +269263.227}
SPL {X  -159.229, Y  +707.508, Z    +0.000, E1   -57.870, E3 +269272.465}
SPL {X  -157.825, Y  +713.519, Z    +0.000, E1   -57.630, E3 +269281.701}
SPL {X  -156.079, Y  +719.864, Z    +0.000, E1   -57.324, E3 +269291.664}
SPL {X  -154.064, Y  +726.175, Z    +0.000, E1   -57.042, E3 +269301.426}
SPL {X  -152.053, Y  +731.726, Z    +0.000, E1   -56.648, E3 +269310.711}
SPL {X  -150.108, Y  +736.570, Z    +0.000, E1   -56.283, E3 +269318.950}
SPL {X  -147.726, Y  +741.964, Z    +0.000, E1   -55.884, E3 +269327.986}
SPL {X  -145.163, Y  +747.242, Z    +0.000, E1   -55.517, E3 +269336.582}
SPL {X  -142.489, Y  +752.286, Z    +0.000, E1   -55.227, E3 +269344.409}
SPL {X  -136.074, Y  +762.910, Z    +0.000, E1   -57.336, E3 +269347.531}
SPL {X  -116.561, Y  +787.183, Z    +0.000, E1   -51.088, E3 +269431.999}
ENDSPLINE

SPLINE
SPL {X  -119.623, Y  +783.957, Z    +0.000, E1   -49.202, E3 +269556.532}
SPL {X  -149.958, Y  +736.927, Z    +0.000, E1   -34.772, E3 +269554.249}
SPL {X  -158.826, Y  +709.343, Z    +0.000, E1   -23.029, E3 +269562.592}
SPL {X  -161.344, Y  +695.370, Z    +0.000, E1   -15.607, E3 +269564.991}
SPL {X  -162.477, Y  +684.065, Z    +0.000, E1    -8.887, E3 +269564.621}
SPL {X  -162.813, Y  +675.055, Z    +0.000, E1    -2.911, E3 +269565.184}
SPL {X  -162.820, Y  +670.901, Z    +0.000, E1    +0.338, E3 +269564.555}
SPL {X  -162.820, Y  +667.984, Z    +0.000, E1    +3.594, E3 +269564.387}
SPL {X  -162.820, Y  +664.667, Z    +0.000, E1    +7.867, E3 +269564.100}
SPL {X  -162.820, Y  +660.022, Z    +0.000, E1   +14.535, E3 +269563.997}
SPL {X  -162.820, Y  +653.408, Z    +0.000, E1   +24.221, E3 +269564.307}
SPL {X  -162.820, Y  +640.244, Z    +0.000, E1   +41.042, E3 +269564.351}
SPL {X  -162.820, Y  +592.517, Z    +0.000, E1   +60.575, E3 +269583.482}
SPL {X  -162.820, Y  +515.613, Z    +0.000, E1   +60.751, E3 +269657.317}
ENDSPLINE

SPLINE
SPL {X  -162.820, Y  +518.198, Z    +0.000, E1   +58.338, E3 +269670.473}
ENDSPLINE

SPLINE
SPL {X  -162.820, Y  +508.314, Z    +0.000, E1   +58.337, E3 +269683.169}
SPL {X  -162.820, Y  +498.518, Z    +0.000, E1   +58.346, E3 +269695.675}
SPL {X  -162.820, Y  +489.418, Z    +0.000, E1   +58.357, E3 +269707.265}
SPL {X  -162.820, Y  +479.904, Z    +0.000, E1   +58.389, E3 +269719.312}
SPL {X  -162.820, Y  +472.095, Z    +0.000, E1   +58.202, E3 +269730.492}
SPL {X  -162.820, Y  +463.661, Z    +0.000, E1   +58.370, E3 +269740.278}
SPL {X  -162.820, Y  +454.904, Z    +0.000, E1   +58.380, E3 +269751.444}
SPL {X  -162.820, Y  +446.206, Z    +0.000, E1   +58.278, E3 +269763.335}
SPL {X  -162.820, Y  +436.416, Z    +0.000, E1   +58.325, E3 +269775.575}
SPL {X  -162.820, Y  +426.628, Z    +0.000, E1   +58.432, E3 +269787.443}
SPL {X  -162.820, Y  +418.389, Z    +0.000, E1   +58.300, E3 +269798.846}
SPL {X  -162.820, Y  +412.292, Z    +0.000, E1   +58.070, E3 +269808.214}
SPL {X  -162.820, Y  +403.663, Z    +0.000, E1   +58.258, E3 +269818.154}
SPL {X  -162.820, Y  +397.157, Z    +0.000, E1   +58.054, E3 +269827.890}
SPL {X  -162.820, Y  +387.359, Z    +0.000, E1   +58.365, E3 +269838.519}
SPL {X  -162.810, Y  +378.731, Z    +0.000, E1   +58.366, E3 +269849.577}
SPL {X  -162.546, Y  +371.051, Z    +0.000, E1   +58.239, E3 +269860.297}
SPL {X  -161.863, Y  +362.875, Z    +0.000, E1   +58.273, E3 +269870.522}
SPL {X  -161.159, Y  +357.301, Z    +0.000, E1   +57.946, E3 +269879.822}
SPL {X  -159.864, Y  +349.614, Z    +0.000, E1   +57.922, E3 +269889.898}
SPL {X  -158.548, Y  +343.449, Z    +0.000, E1   +57.711, E3 +269899.072}
SPL {X  -156.580, Y  +335.856, Z    +0.000, E1   +57.340, E3 +269911.295}
SPL {X  -154.237, Y  +328.333, Z    +0.000, E1   +56.930, E3 +269923.214}
SPL {X  -152.732, Y  +324.078, Z    +0.000, E1   +56.482, E3 +269931.219}
SPL {X  -150.609, Y  +318.634, Z    +0.000, E1   +56.366, E3 +269938.913}
SPL {X  -148.206, Y  +313.080, Z    +0.000, E1   +55.888, E3 +269948.625}
SPL {X  -145.956, Y  +308.339, Z    +0.000, E1   +55.380, E3 +269957.301}
SPL {X  -142.234, Y  +301.255, Z    +0.000, E1   +55.418, E3 +269966.175}
SPL {X  -134.491, Y  +288.726, Z    +0.000, E1   +57.448, E3 +269971.831}
SPL {X  -115.845, Y  +266.087, Z    +0.000, E1   +50.276, E3 +270068.442}
SPL {X  -114.083, Y  +264.330, Z    +0.000, E1   +49.123, E3 +270107.152}
ENDSPLINE

SPLINE
SPL {X  -136.188, Y  +291.263, Z    +0.000, E1   +45.457, E3 +270203.218}
SPL {X  -151.738, Y  +321.457, Z    +0.000, E1   +32.773, E3 +270170.387}
SPL {X  -158.704, Y  +344.121, Z    +0.000, E1   +23.312, E3 +270185.537}
SPL {X  -162.109, Y  +365.304, Z    +0.000, E1   +11.761, E3 +270184.839}
SPL {X  -162.811, Y  +378.776, Z    +0.000, E1    +3.078, E3 +270185.083}
SPL {X  -162.820, Y  +383.454, Z    +0.000, E1    -0.619, E3 +270184.551}
SPL {X  -162.820, Y  +387.033, Z    +0.000, E1    -4.758, E3 +270184.255}
SPL {X  -162.820, Y  +390.967, Z    +0.000, E1    -9.918, E3 +270184.700}
SPL {X  -162.820, Y  +395.392, Z    +0.000, E1   -16.726, E3 +270183.141}
SPL {X  -162.820, Y  +402.654, Z    +0.000, E1   -26.492, E3 +270185.032}
SPL {X  -162.820, Y  +417.515, Z    +0.000, E1   -44.878, E3 +270184.149}
SPL {X  -162.820, Y  +462.065, Z    +0.000, E1   -61.507, E3 +270201.109}
SPL {X  -162.820, Y  +504.602, Z    +0.000, E1   -64.286, E3 +270226.635}
SPL {X  -162.820, Y  +539.530, Z    +0.000, E1   -60.821, E3 +270277.326}
ENDSPLINE

SPLINE
SPL {X  -162.820, Y  +534.172, Z    +0.000, E1   -58.470, E3 +270286.826}
ENDSPLINE

SPLINE
SPL {X  -162.820, Y  +543.678, Z    +0.000, E1   -58.515, E3 +270298.703}
SPL {X  -162.820, Y  +553.725, Z    +0.000, E1   -58.454, E3 +270311.964}
SPL {X  -162.820, Y  +562.850, Z    +0.000, E1   -58.373, E3 +270324.126}
SPL {X  -162.820, Y  +571.217, Z    +0.000, E1   -58.397, E3 +270334.679}
SPL {X  -162.820, Y  +581.879, Z    +0.000, E1   -58.475, E3 +270347.932}
SPL {X  -162.820, Y  +591.768, Z    +0.000, E1   -58.375, E3 +270361.130}
SPL {X  -162.820, Y  +601.090, Z    +0.000, E1   -58.519, E3 +270372.117}
SPL {X  -162.820, Y  +609.492, Z    +0.000, E1   -58.431, E3 +270383.422}
SPL {X  -162.820, Y  +617.241, Z    +0.000, E1   -58.340, E3 +270393.947}
SPL {X  -162.820, Y  +626.506, Z    +0.000, E1   -58.420, E3 +270405.329}
SPL {X  -162.820, Y  +635.919, Z    +0.000, E1   -58.604, E3 +270416.073}
SPL {X  -162.820, Y  +643.895, Z    +0.000, E1   -58.380, E3 +270427.838}
SPL {X  -162.820, Y  +653.118, Z    +0.000, E1   -58.401, E3 +270439.435}
SPL {X  -162.820, Y  +660.924, Z    +0.000, E1   -58.393, E3 +270449.503}
SPL {X  -162.820, Y  +670.459, Z    +0.000, E1   -58.489, E3 +270461.104}
SPL {X  -162.713, Y  +679.396, Z    +0.000, E1   -58.414, E3 +270473.003}
SPL {X  -162.301, Y  +686.495, Z    +0.000, E1   -58.302, E3 +270482.787}
SPL {X  -161.571, Y  +693.631, Z    +0.000, E1   -58.186, E3 +270492.751}
SPL {X  -160.411, Y  +701.402, Z    +0.000, E1   -58.100, E3 +270503.227}
SPL {X  -159.229, Y  +707.508, Z    +0.000, E1   -57.870, E3 +270512.465}
SPL {X  -157.825, Y  +713.519, Z    +0.000, E1   -57.630, E3 +270521.701}
SPL {X  -156.079, Y  +719.864, Z    +0.000, E1   -57.324, E3 +270531.664}
SPL {X  -154.064, Y  +726.175, Z    +0.000, E1   -57.042, E3 +270541.426}
SPL {X  -152.053, Y  +731.726, Z    +0.000, E1   -56.648, E3 +270550.711}
SPL {X  -150.108, Y  +736.570, Z    +0.000, E1   -56.283, E3 +270558.950}
SPL {X  -147.726, Y  +741.964, Z    +0.000, E1   -55.884, E3 +270567.986}
SPL {X  -145.163, Y  +747.242, Z    +0.000, E1   -55.517, E3 +270576.582}
SPL {X  -142.489, Y  +752.286, Z    +0.000, E1   -55.227, E3 +270584.409}
SPL {X  -136.074, Y  +762.910, Z    +0.000, E1   -57.336, E3 +270587.531}
SPL {X  -121.244, Y  +782.175, Z    +0.000, E1   -51.023, E3 +270659.476}
SPL {X  -114.422, Y  +789.335, Z    +0.000, E1   -51.094, E3 +270678.092}
ENDSPLINE

SPLINE
SPL {X  -119.623, Y  +783.957, Z    +0.000, E1   -49.202, E3 +270796.532}
SPL {X  -149.958, Y  +736.927, Z    +0.000, E1   -34.772, E3 +270794.249}
SPL {X  -158.826, Y  +709.343, Z    +0.000, E1   -23.029, E3 +270802.592}
SPL {X  -161.800, Y  +691.694, Z    +0.000, E1   -13.520, E3 +270804.886}
SPL {X  -162.597, Y  +682.022, Z    +0.000, E1    -7.544, E3 +270804.542}
SPL {X  -162.813, Y  +675.055, Z    +0.000, E1    -2.911, E3 +270805.184}
SPL {X  -162.820, Y  +670.901, Z    +0.000, E1    +0.338, E3 +270804.555}
SPL {X  -162.820, Y  +667.984, Z    +0.000, E1    +3.594, E3 +270804.387}
SPL {X  -162.820, Y  +664.667, Z    +0.000, E1    +7.867, E3 +270804.100}
SPL {X  -162.820, Y  +660.022, Z    +0.000, E1   +14.535, E3 +270803.997}
SPL {X  -162.820, Y  +653.408, Z    +0.000, E1   +24.221, E3 +270804.307}
SPL {X  -162.820, Y  +640.244, Z    +0.000, E1   +41.042, E3 +270804.351}
SPL {X  -162.820, Y  +602.578, Z    +0.000, E1   +60.061, E3 +270815.766}
SPL {X  -162.820, Y  +586.468, Z    +0.000, E1   +60.779, E3 +270828.168}
SPL {X  -162.820, Y  +515.613, Z    +0.000, E1   +60.751, E3 +270897.317}
ENDSPLINE

SPLINE
SPL {X  -162.820, Y  +518.198, Z    +0.000, E1   +58.338, E3 +270910.473}
ENDSPLINE

SPLINE
SPL {X  -162.820, Y  +508.314, Z    +0.000, E1   +58.337, E3 +270923.169}
SPL {X  -162.820, Y  +498.518, Z    +0.000, E1   +58.346, E3 +270935.675}
SPL {X  -162.820, Y  +489.418, Z    +0.000, E1   +58.357, E3 +270947.265}
SPL {X  -162.820, Y  +479.904, Z    +0.000, E1   +58.389, E3 +270959.312}
SPL {X  -162.820, Y  +472.095, Z    +0.000, E1   +58.202, E3 +270970.492}
SPL {X  -162.820, Y  +463.661, Z    +0.000, E1   +58.370, E3 +270980.278}
SPL {X  -162.820, Y  +454.904, Z    +0.000, E1   +58.380, E3 +270991.444}
SPL {X  -162.820, Y  +446.206, Z    +0.000, E1   +58.278, E3 +271003.335}
SPL {X  -162.820, Y  +436.416, Z    +0.000, E1   +58.325, E3 +271015.575}
SPL {X  -162.820, Y  +426.628, Z    +0.000, E1   +58.432, E3 +271027.443}
SPL {X  -162.820, Y  +418.389, Z    +0.000, E1   +58.300, E3 +271038.846}
SPL {X  -162.820, Y  +412.292, Z    +0.000, E1   +58.070, E3 +271048.214}
SPL {X  -162.820, Y  +403.663, Z    +0.000, E1   +58.258, E3 +271058.154}
ENDSPLINE

SPLINE
SPL {X  -162.820, Y  +411.119, Z    +0.000, E1   +54.525, E3 +271072.194}
ENDSPLINE

SPLINE
SPL {X  -162.820, Y  +400.244, Z    +0.000, E1   +54.630, E3 +271087.546}
SPL {X  -162.820, Y  +389.249, Z    +0.000, E1   +54.752, E3 +271103.125}
SPL {X  -162.799, Y  +377.862, Z    +0.000, E1   +54.622, E3 +271120.756}
SPL {X  -162.373, Y  +368.447, Z    +0.000, E1   +54.597, E3 +271134.684}
SPL {X  -161.939, Y  +363.587, Z    +0.000, E1   +54.355, E3 +271143.297}
SPL {X  -160.880, Y  +355.442, Z    +0.000, E1   +54.372, E3 +271155.508}
SPL {X  -159.457, Y  +347.579, Z    +0.000, E1   +54.148, E3 +271168.244}
SPL {X  -158.033, Y  +341.310, Z    +0.000, E1   +53.819, E3 +271179.581}
SPL {X  -156.195, Y  +334.528, Z    +0.000, E1   +53.534, E3 +271191.146}
SPL {X  -154.120, Y  +327.988, Z    +0.000, E1   +53.171, E3 +271203.003}
SPL {X  -151.310, Y  +320.369, Z    +0.000, E1   +52.706, E3 +271216.718}
SPL {X  -148.923, Y  +314.679, Z    +0.000, E1   +52.172, E3 +271227.803}
SPL {X  -146.846, Y  +310.168, Z    +0.000, E1   +51.697, E3 +271236.864}
SPL {X  -140.627, Y  +298.437, Z    +0.000, E1   +54.251, E3 +271241.123}
SPL {X  -122.064, Y  +272.747, Z    +0.000, E1   +48.156, E3 +271346.648}
ENDSPLINE

SPLINE
SPL {X  -148.173, Y  +313.009, Z    +0.000, E1   +35.624, E3 +271429.694}
SPL {X  -159.343, Y  +347.032, Z    +0.000, E1   +21.245, E3 +271433.537}
SPL {X  -161.787, Y  +362.186, Z    +0.000, E1   +13.182, E3 +271434.733}
SPL {X  -162.692, Y  +374.052, Z    +0.000, E1    +6.208, E3 +271434.579}
SPL {X  -162.820, Y  +382.143, Z    +0.000, E1    +0.693, E3 +271434.714}
SPL {X  -162.820, Y  +385.887, Z    +0.000, E1    -2.819, E3 +271434.386}
SPL {X  -162.820, Y  +389.383, Z    +0.000, E1    -6.871, E3 +271434.453}
SPL {X  -162.820, Y  +393.153, Z    +0.000, E1   -11.600, E3 +271434.346}
SPL {X  -162.820, Y  +400.748, Z    +0.000, E1   -21.791, E3 +271434.138}
SPL {X  -162.820, Y  +413.615, Z    +0.000, E1   -37.560, E3 +271434.232}
SPL {X  -162.820, Y  +456.390, Z    +0.000, E1   -57.415, E3 +271451.273}
SPL {X  -162.820, Y  +525.017, Z    +0.000, E1   -58.379, E3 +271521.938}
ENDSPLINE

SPLINE
SPL {X  -162.820, Y  +520.266, Z    +0.000, E1   -55.155, E3 +271536.431}
ENDSPLINE

SPLINE
SPL {X  -162.820, Y  +529.742, Z    +0.000, E1   -55.146, E3 +271550.147}
SPL {X  -162.820, Y  +538.383, Z    +0.000, E1   -55.306, E3 +271561.599}
SPL {X  -162.820, Y  +544.790, Z    +0.000, E1   -55.066, E3 +271572.399}
SPL {X  -162.820, Y  +552.981, Z    +0.000, E1   -55.286, E3 +271582.862}
SPL {X  -162.820, Y  +560.767, Z    +0.000, E1   -55.137, E3 +271595.170}
SPL {X  -162.820, Y  +570.590, Z    +0.000, E1   -55.270, E3 +271608.504}
SPL {X  -162.820, Y  +580.865, Z    +0.000, E1   -55.132, E3 +271624.461}
SPL {X  -162.820, Y  +594.246, Z    +0.000, E1   -55.310, E3 +271642.660}
SPL {X  -162.820, Y  +601.811, Z    +0.000, E1   -55.027, E3 +271655.187}
SPL {X  -162.820, Y  +609.951, Z    +0.000, E1   -55.211, E3 +271665.934}
SPL {X  -162.820, Y  +618.960, Z    +0.000, E1   -55.186, E3 +271679.154}
SPL {X  -162.820, Y  +627.322, Z    +0.000, E1   -55.201, E3 +271691.089}
SPL {X  -162.820, Y  +634.693, Z    +0.000, E1   -55.198, E3 +271701.806}
SPL {X  -162.820, Y  +642.452, Z    +0.000, E1   -55.141, E3 +271713.413}
SPL {X  -162.820, Y  +649.370, Z    +0.000, E1   -55.160, E3 +271723.270}
SPL {X  -162.820, Y  +658.542, Z    +0.000, E1   -55.251, E3 +271736.148}
SPL {X  -162.820, Y  +671.259, Z    +0.000, E1   -55.266, E3 +271754.525}
SPL {X  -162.498, Y  +683.731, Z    +0.000, E1   -55.157, E3 +271773.235}
SPL {X  -161.784, Y  +691.841, Z    +0.000, E1   -55.010, E3 +271785.691}
SPL {X  -161.070, Y  +697.305, Z    +0.000, E1   -54.828, E3 +271794.769}
SPL {X  -159.751, Y  +704.965, Z    +0.000, E1   -54.697, E3 +271806.755}
SPL {X  -158.271, Y  +711.718, Z    +0.000, E1   -54.504, E3 +271817.564}
SPL {X  -157.115, Y  +716.223, Z    +0.000, E1   -54.227, E3 +271825.756}
SPL {X  -154.825, Y  +723.894, Z    +0.000, E1   -53.830, E3 +271839.296}
SPL {X  -152.160, Y  +731.445, Z    +0.000, E1   -53.336, E3 +271852.838}
SPL {X  -150.059, Y  +736.687, Z    +0.000, E1   -53.023, E3 +271862.004}
SPL {X  -147.746, Y  +741.922, Z    +0.000, E1   -52.631, E3 +271871.711}
SPL {X  -144.373, Y  +748.778, Z    +0.000, E1   -52.887, E3 +271880.124}
SPL {X  -137.947, Y  +759.993, Z    +0.000, E1   -55.381, E3 +271883.234}
SPL {X  -123.111, Y  +780.056, Z    +0.000, E1   -48.144, E3 +271982.369}
ENDSPLINE

SPLINE
SPL {X  -146.599, Y  +744.345, Z    +0.000, E1   -36.661, E3 +272067.373}
SPL {X  -157.185, Y  +715.965, Z    +0.000, E1   -25.340, E3 +272070.422}
SPL {X  -159.997, Y  +703.690, Z    +0.000, E1   -19.457, E3 +272071.751}
SPL {X  -161.886, Y  +690.913, Z    +0.000, E1   -12.672, E3 +272075.879}
SPL {X  -162.700, Y  +679.756, Z    +0.000, E1    -6.060, E3 +272075.088}
SPL {X  -162.820, Y  +673.439, Z    +0.000, E1    -1.797, E3 +272075.190}
SPL {X  -162.820, Y  +670.554, Z    +0.000, E1    +0.472, E3 +272074.722}
SPL {X  -162.820, Y  +667.789, Z    +0.000, E1    +3.144, E3 +272074.744}
SPL {X  -162.820, Y  +664.083, Z    +0.000, E1    +7.387, E3 +272074.636}
SPL {X  -162.820, Y  +659.344, Z    +0.000, E1   +13.535, E3 +272074.199}
SPL {X  -162.820, Y  +653.403, Z    +0.000, E1   +21.415, E3 +272074.614}
SPL {X  -162.820, Y  +642.162, Z    +0.000, E1   +35.510, E3 +272073.926}
SPL {X  -162.820, Y  +598.675, Z    +0.000, E1   +56.845, E3 +272091.239}
SPL {X  -162.820, Y  +542.287, Z    +0.000, E1   +54.257, E3 +272170.143}
SPL {X  -162.820, Y  +533.839, Z    +0.000, E1   +53.682, E3 +272186.563}
SPL {X  -162.820, Y  +525.300, Z    +0.000, E1   +53.701, E3 +272199.339}
SPL {X  -162.820, Y  +518.365, Z    +0.000, E1   +53.683, E3 +272210.132}
SPL {X  -162.820, Y  +510.654, Z    +0.000, E1   +53.658, E3 +272222.131}
SPL {X  -162.820, Y  +501.304, Z    +0.000, E1   +53.758, E3 +272235.820}
SPL {X  -162.820, Y  +493.008, Z    +0.000, E1   +53.586, E3 +272249.595}
SPL {X  -162.820, Y  +485.759, Z    +0.000, E1   +53.138, E3 +272263.603}
ENDSPLINE

SPLINE
SPL {X  -162.820, Y  +494.645, Z    +0.000, E1   +48.544, E3 +272276.078}
ENDSPLINE

SPLINE
SPL {X  -162.820, Y  +486.578, Z    +0.000, E1   +49.194, E3 +272286.875}
SPL {X  -162.820, Y  +476.731, Z    +0.000, E1   +50.039, E3 +272299.298}
SPL {X  -162.820, Y  +466.442, Z    +0.000, E1   +50.873, E3 +272311.966}
SPL {X  -162.820, Y  +455.624, Z    +0.000, E1   +51.698, E3 +272325.037}
SPL {X  -162.820, Y  +444.568, Z    +0.000, E1   +52.608, E3 +272337.350}
SPL {X  -162.820, Y  +432.435, Z    +0.000, E1   +53.605, E3 +272350.233}
SPL {X  -162.820, Y  +419.900, Z    +0.000, E1   +54.598, E3 +272362.908}
SPL {X  -162.820, Y  +411.092, Z    +0.000, E1   +54.552, E3 +272376.428}
SPL {X  -162.820, Y  +400.244, Z    +0.000, E1   +54.630, E3 +272391.894}
SPL {X  -162.820, Y  +389.249, Z    +0.000, E1   +54.752, E3 +272407.473}
SPL {X  -162.799, Y  +377.862, Z    +0.000, E1   +54.622, E3 +272425.104}
SPL {X  -162.373, Y  +368.447, Z    +0.000, E1   +54.597, E3 +272439.032}
SPL {X  -161.939, Y  +363.587, Z    +0.000, E1   +54.355, E3 +272447.645}
SPL {X  -161.062, Y  +356.641, Z    +0.000, E1   +54.440, E3 +272457.517}
SPL {X  -159.761, Y  +349.086, Z    +0.000, E1   +54.132, E3 +272470.539}
SPL {X  -158.451, Y  +343.033, Z    +0.000, E1   +53.828, E3 +272481.215}
SPL {X  -156.619, Y  +335.993, Z    +0.000, E1   +53.639, E3 +272492.861}
SPL {X  -154.959, Y  +330.520, Z    +0.000, E1   +53.198, E3 +272503.287}
SPL {X  -153.385, Y  +325.878, Z    +0.000, E1   +53.068, E3 +272510.868}
SPL {X  -151.310, Y  +320.369, Z    +0.000, E1   +52.706, E3 +272521.066}
SPL {X  -148.923, Y  +314.679, Z    +0.000, E1   +52.172, E3 +272532.151}
SPL {X  -146.846, Y  +310.168, Z    +0.000, E1   +51.697, E3 +272541.212}
SPL {X  -140.627, Y  +298.437, Z    +0.000, E1   +54.251, E3 +272545.470}
SPL {X  -122.064, Y  +272.747, Z    +0.000, E1   +48.156, E3 +272650.996}
ENDSPLINE

SPLINE
SPL {X  -148.173, Y  +313.009, Z    +0.000, E1   +35.624, E3 +272734.041}
SPL {X  -159.343, Y  +347.032, Z    +0.000, E1   +21.245, E3 +272737.885}
SPL {X  -162.355, Y  +368.197, Z    +0.000, E1    +9.799, E3 +272739.054}
SPL {X  -162.819, Y  +380.071, Z    +0.000, E1    +2.240, E3 +272739.048}
SPL {X  -162.820, Y  +383.414, Z    +0.000, E1    -0.499, E3 +272739.011}
SPL {X  -162.820, Y  +385.887, Z    +0.000, E1    -2.819, E3 +272738.734}
SPL {X  -162.820, Y  +389.383, Z    +0.000, E1    -6.871, E3 +272738.801}
SPL {X  -162.820, Y  +393.153, Z    +0.000, E1   -11.600, E3 +272738.694}
SPL {X  -162.820, Y  +400.748, Z    +0.000, E1   -21.791, E3 +272738.486}
SPL {X  -162.820, Y  +413.615, Z    +0.000, E1   -37.560, E3 +272738.580}
SPL {X  -162.820, Y  +456.390, Z    +0.000, E1   -57.415, E3 +272755.621}
SPL {X  -162.820, Y  +525.017, Z    +0.000, E1   -58.379, E3 +272826.286}
ENDSPLINE

SPLINE
SPL {X  -162.820, Y  +520.266, Z    +0.000, E1   -55.155, E3 +272840.779}
ENDSPLINE

SPLINE
SPL {X  -162.820, Y  +529.742, Z    +0.000, E1   -55.146, E3 +272854.495}
SPL {X  -162.820, Y  +538.383, Z    +0.000, E1   -55.306, E3 +272865.947}
SPL {X  -162.820, Y  +544.790, Z    +0.000, E1   -55.066, E3 +272876.747}
SPL {X  -162.820, Y  +552.981, Z    +0.000, E1   -55.286, E3 +272887.209}
SPL {X  -162.820, Y  +560.767, Z    +0.000, E1   -55.137, E3 +272899.518}
SPL {X  -162.820, Y  +570.590, Z    +0.000, E1   -55.270, E3 +272912.852}
SPL {X  -162.820, Y  +577.946, Z    +0.000, E1   -55.110, E3 +272924.490}
SPL {X  -162.820, Y  +583.981, Z    +0.000, E1   -55.057, E3 +272933.572}
SPL {X  -162.820, Y  +594.246, Z    +0.000, E1   -55.310, E3 +272947.007}
SPL {X  -162.820, Y  +601.811, Z    +0.000, E1   -55.027, E3 +272959.535}
SPL {X  -162.820, Y  +609.951, Z    +0.000, E1   -55.211, E3 +272970.282}
SPL {X  -162.820, Y  +618.960, Z    +0.000, E1   -55.186, E3 +272983.502}
SPL {X  -162.820, Y  +627.322, Z    +0.000, E1   -55.201, E3 +272995.437}
SPL {X  -162.820, Y  +634.693, Z    +0.000, E1   -55.198, E3 +273006.154}
SPL {X  -162.820, Y  +642.452, Z    +0.000, E1   -55.141, E3 +273017.761}
SPL {X  -162.820, Y  +652.837, Z    +0.000, E1   -55.281, E3 +273032.028}
SPL {X  -162.820, Y  +660.849, Z    +0.000, E1   -55.101, E3 +273044.577}
SPL {X  -162.820, Y  +668.534, Z    +0.000, E1   -55.182, E3 +273055.291}
SPL {X  -162.763, Y  +677.803, Z    +0.000, E1   -55.175, E3 +273068.797}
SPL {X  -162.084, Y  +688.960, Z    +0.000, E1   -55.150, E3 +273085.252}
SPL {X  -161.070, Y  +697.305, Z    +0.000, E1   -54.828, E3 +273099.117}
SPL {X  -159.751, Y  +704.965, Z    +0.000, E1   -54.697, E3 +273111.103}
SPL {X  -158.271, Y  +711.718, Z    +0.000, E1   -54.504, E3 +273121.912}
SPL {X  -157.115, Y  +716.223, Z    +0.000, E1   -54.227, E3 +273130.103}
SPL {X  -155.622, Y  +721.376, Z    +0.000, E1   -53.849, E3 +273139.703}
SPL {X  -153.323, Y  +728.294, Z    +0.000, E1   -53.618, E3 +273151.176}
SPL {X  -150.606, Y  +735.372, Z    +0.000, E1   -53.091, E3 +273164.173}
SPL {X  -148.712, Y  +739.795, Z    +0.000, E1   -52.656, E3 +273172.736}
SPL {X  -146.885, Y  +743.751, Z    +0.000, E1   -52.544, E3 +273179.009}
SPL {X  -144.373, Y  +748.778, Z    +0.000, E1   -52.887, E3 +273184.472}
SPL {X  -137.947, Y  +759.993, Z    +0.000, E1   -55.381, E3 +273187.581}
SPL {X  -123.111, Y  +780.056, Z    +0.000, E1   -48.144, E3 +273286.717}
ENDSPLINE

SPLINE
SPL {X  -146.599, Y  +744.345, Z    +0.000, E1   -36.661, E3 +273371.720}
SPL {X  -158.886, Y  +709.076, Z    +0.000, E1   -22.176, E3 +273375.592}
SPL {X  -161.886, Y  +690.913, Z    +0.000, E1   -12.672, E3 +273380.227}
SPL {X  -162.573, Y  +682.458, Z    +0.000, E1    -7.683, E3 +273379.728}
SPL {X  -162.817, Y  +674.426, Z    +0.000, E1    -2.573, E3 +273379.446}
SPL {X  -162.820, Y  +670.554, Z    +0.000, E1    +0.472, E3 +273379.070}
SPL {X  -162.820, Y  +667.789, Z    +0.000, E1    +3.144, E3 +273379.092}
SPL {X  -162.820, Y  +664.083, Z    +0.000, E1    +7.387, E3 +273378.983}
SPL {X  -162.820, Y  +659.344, Z    +0.000, E1   +13.535, E3 +273378.547}
SPL {X  -162.820, Y  +653.403, Z    +0.000, E1   +21.415, E3 +273378.962}
SPL {X  -162.820, Y  +642.162, Z    +0.000, E1   +35.510, E3 +273378.274}
SPL {X  -162.820, Y  +598.675, Z    +0.000, E1   +56.845, E3 +273395.587}
SPL {X  -162.820, Y  +543.175, Z    +0.000, E1   +54.504, E3 +273471.441}
SPL {X  -162.820, Y  +538.115, Z    +0.000, E1   +53.658, E3 +273484.493}
SPL {X  -162.820, Y  +527.429, Z    +0.000, E1   +53.760, E3 +273500.222}
SPL {X  -162.820, Y  +518.365, Z    +0.000, E1   +53.683, E3 +273514.480}
SPL {X  -162.820, Y  +510.654, Z    +0.000, E1   +53.658, E3 +273526.479}
SPL {X  -162.820, Y  +501.304, Z    +0.000, E1   +53.758, E3 +273540.168}
SPL {X  -162.820, Y  +493.008, Z    +0.000, E1   +53.586, E3 +273553.943}
SPL {X  -162.820, Y  +484.615, Z    +0.000, E1   +53.726, E3 +273565.874}
ENDSPLINE

SPLINE
SPL {X  -162.820, Y  +492.996, Z    +0.000, E1   +49.430, E3 +273578.420}
ENDSPLINE

SPLINE
SPL {X  -162.820, Y  +486.578, Z    +0.000, E1   +49.194, E3 +273591.222}
SPL {X  -162.820, Y  +476.731, Z    +0.000, E1   +50.039, E3 +273603.645}
SPL {X  -162.820, Y  +466.442, Z    +0.000, E1   +50.873, E3 +273616.314}
SPL {X  -162.820, Y  +455.624, Z    +0.000, E1   +51.698, E3 +273629.385}
SPL {X  -162.820, Y  +444.568, Z    +0.000, E1   +52.608, E3 +273641.698}
SPL {X  -162.820, Y  +432.435, Z    +0.000, E1   +53.605, E3 +273654.581}
SPL {X  -162.820, Y  +419.900, Z    +0.000, E1   +54.598, E3 +273667.255}
SPL {X  -162.820, Y  +411.092, Z    +0.000, E1   +54.552, E3 +273680.775}
SPL {X  -162.820, Y  +400.244, Z    +0.000, E1   +54.630, E3 +273696.242}
SPL {X  -162.820, Y  +389.249, Z    +0.000, E1   +54.752, E3 +273711.821}
SPL {X  -162.820, Y  +380.650, Z    +0.000, E1   +54.601, E3 +273725.266}
SPL {X  -162.727, Y  +374.992, Z    +0.000, E1   +54.549, E3 +273733.948}
SPL {X  -162.216, Y  +366.490, Z    +0.000, E1   +54.549, E3 +273746.747}
SPL {X  -161.062, Y  +356.641, Z    +0.000, E1   +54.440, E3 +273761.865}
SPL {X  -159.761, Y  +349.086, Z    +0.000, E1   +54.132, E3 +273774.886}
SPL {X  -158.033, Y  +341.310, Z    +0.000, E1   +53.819, E3 +273788.276}
SPL {X  -156.195, Y  +334.528, Z    +0.000, E1   +53.534, E3 +273799.842}
SPL {X  -154.120, Y  +327.988, Z    +0.000, E1   +53.171, E3 +273811.699}
SPL {X  -151.310, Y  +320.369, Z    +0.000, E1   +52.706, E3 +273825.414}
SPL {X  -148.923, Y  +314.679, Z    +0.000, E1   +52.172, E3 +273836.498}
SPL {X  -146.846, Y  +310.168, Z    +0.000, E1   +51.697, E3 +273845.559}
SPL {X  -140.627, Y  +298.437, Z    +0.000, E1   +54.251, E3 +273849.818}
SPL {X  -122.064, Y  +272.747, Z    +0.000, E1   +48.156, E3 +273955.344}
ENDSPLINE

SPLINE
SPL {X  -148.173, Y  +313.009, Z    +0.000, E1   +35.624, E3 +274038.389}
SPL {X  -158.289, Y  +342.356, Z    +0.000, E1   +23.452, E3 +274041.379}
SPL {X  -161.301, Y  +358.312, Z    +0.000, E1   +15.384, E3 +274043.336}
SPL {X  -162.692, Y  +374.052, Z    +0.000, E1    +6.208, E3 +274043.275}
SPL {X  -162.820, Y  +381.030, Z    +0.000, E1    +1.454, E3 +274043.453}
SPL {X  -162.820, Y  +384.274, Z    +0.000, E1    -1.205, E3 +274043.173}
SPL {X  -162.820, Y  +388.271, Z    +0.000, E1    -5.458, E3 +274043.165}
SPL {X  -162.820, Y  +394.827, Z    +0.000, E1   -13.677, E3 +274042.855}
SPL {X  -162.820, Y  +402.977, Z    +0.000, E1   -24.772, E3 +274043.137}
SPL {X  -162.820, Y  +413.615, Z    +0.000, E1   -37.560, E3 +274042.928}
SPL {X  -162.820, Y  +456.390, Z    +0.000, E1   -57.415, E3 +274059.969}
SPL {X  -162.820, Y  +525.017, Z    +0.000, E1   -58.379, E3 +274130.634}
ENDSPLINE

SPLINE
SPL {X  -162.820, Y  +515.796, Z    +0.000, E1   -54.952, E3 +274139.740}
ENDSPLINE

SPLINE
SPL {X  -162.820, Y  +522.537, Z    +0.000, E1   -55.218, E3 +274147.915}
SPL {X  -162.820, Y  +529.742, Z    +0.000, E1   -55.146, E3 +274158.842}
SPL {X  -162.820, Y  +538.383, Z    +0.000, E1   -55.306, E3 +274170.295}
SPL {X  -162.820, Y  +544.790, Z    +0.000, E1   -55.066, E3 +274181.095}
SPL {X  -162.820, Y  +552.981, Z    +0.000, E1   -55.286, E3 +274191.557}
SPL {X  -162.820, Y  +560.767, Z    +0.000, E1   -55.137, E3 +274203.866}
SPL {X  -162.820, Y  +570.590, Z    +0.000, E1   -55.270, E3 +274217.200}
SPL {X  -162.820, Y  +577.946, Z    +0.000, E1   -55.110, E3 +274228.837}
SPL {X  -162.820, Y  +583.981, Z    +0.000, E1   -55.057, E3 +274237.920}
SPL {X  -162.820, Y  +591.604, Z    +0.000, E1   -55.202, E3 +274248.094}
SPL {X  -162.820, Y  +600.465, Z    +0.000, E1   -55.218, E3 +274260.882}
SPL {X  -162.820, Y  +609.951, Z    +0.000, E1   -55.211, E3 +274274.630}
SPL {X  -162.820, Y  +617.278, Z    +0.000, E1   -55.256, E3 +274284.854}
SPL {X  -162.820, Y  +625.209, Z    +0.000, E1   -55.167, E3 +274297.046}
SPL {X  -162.820, Y  +634.693, Z    +0.000, E1   -55.198, E3 +274310.502}
SPL {X  -162.820, Y  +642.452, Z    +0.000, E1   -55.141, E3 +274322.108}
SPL {X  -162.820, Y  +652.837, Z    +0.000, E1   -55.281, E3 +274336.376}
SPL {X  -162.820, Y  +660.849, Z    +0.000, E1   -55.101, E3 +274348.925}
SPL {X  -162.820, Y  +668.534, Z    +0.000, E1   -55.182, E3 +274359.639}
SPL {X  -162.763, Y  +677.803, Z    +0.000, E1   -55.175, E3 +274373.145}
SPL {X  -162.314, Y  +686.325, Z    +0.000, E1   -55.173, E3 +274385.425}
SPL {X  -161.784, Y  +691.841, Z    +0.000, E1   -55.010, E3 +274394.387}
SPL {X  -161.070, Y  +697.305, Z    +0.000, E1   -54.828, E3 +274403.465}
SPL {X  -159.751, Y  +704.965, Z    +0.000, E1   -54.697, E3 +274415.451}
SPL {X  -158.271, Y  +711.718, Z    +0.000, E1   -54.504, E3 +274426.260}
SPL {X  -157.115, Y  +716.223, Z    +0.000, E1   -54.227, E3 +274434.451}
SPL {X  -155.622, Y  +721.376, Z    +0.000, E1   -53.849, E3 +274444.051}
SPL {X  -153.323, Y  +728.294, Z    +0.000, E1   -53.618, E3 +274455.524}
SPL {X  -150.606, Y  +735.372, Z    +0.000, E1   -53.091, E3 +274468.521}
SPL {X  -148.712, Y  +739.795, Z    +0.000, E1   -52.656, E3 +274477.084}
SPL {X  -146.885, Y  +743.751, Z    +0.000, E1   -52.544, E3 +274483.357}
SPL {X  -144.373, Y  +748.778, Z    +0.000, E1   -52.887, E3 +274488.820}
SPL {X  -137.947, Y  +759.993, Z    +0.000, E1   -55.381, E3 +274491.929}
SPL {X  -123.111, Y  +780.056, Z    +0.000, E1   -48.144, E3 +274591.065}
ENDSPLINE

SPLINE
SPL {X  -146.599, Y  +744.345, Z    +0.000, E1   -36.661, E3 +274676.068}
SPL {X  -158.886, Y  +709.076, Z    +0.000, E1   -22.176, E3 +274679.940}
SPL {X  -161.886, Y  +690.913, Z    +0.000, E1   -12.672, E3 +274684.575}
SPL {X  -162.573, Y  +682.458, Z    +0.000, E1    -7.683, E3 +274684.076}
SPL {X  -162.817, Y  +674.426, Z    +0.000, E1    -2.573, E3 +274683.794}
SPL {X  -162.820, Y  +670.554, Z    +0.000, E1    +0.472, E3 +274683.418}
SPL {X  -162.820, Y  +667.789, Z    +0.000, E1    +3.144, E3 +274683.440}
SPL {X  -162.820, Y  +664.083, Z    +0.000, E1    +7.387, E3 +274683.331}
SPL {X  -162.820, Y  +659.344, Z    +0.000, E1   +13.535, E3 +274682.895}
SPL {X  -162.820, Y  +653.403, Z    +0.000, E1   +21.415, E3 +274683.310}
SPL {X  -162.820, Y  +644.970, Z    +0.000, E1   +32.346, E3 +274682.726}
SPL {X  -162.820, Y  +637.013, Z    +0.000, E1   +41.185, E3 +274682.431}
SPL {X  -162.820, Y  +603.840, Z    +0.000, E1   +55.833, E3 +274697.048}
SPL {X  -162.820, Y  +590.612, Z    +0.000, E1   +58.217, E3 +274704.432}
SPL {X  -162.820, Y  +543.175, Z    +0.000, E1   +54.504, E3 +274775.789}
SPL {X  -162.820, Y  +538.115, Z    +0.000, E1   +53.658, E3 +274788.840}
SPL {X  -162.820, Y  +530.332, Z    +0.000, E1   +53.757, E3 +274799.983}
SPL {X  -162.820, Y  +525.300, Z    +0.000, E1   +53.701, E3 +274808.034}
SPL {X  -162.820, Y  +518.365, Z    +0.000, E1   +53.683, E3 +274818.828}
SPL {X  -162.820, Y  +508.465, Z    +0.000, E1   +53.706, E3 +274834.043}
SPL {X  -162.820, Y  +499.206, Z    +0.000, E1   +53.779, E3 +274847.482}
SPL {X  -162.820, Y  +493.008, Z    +0.000, E1   +53.586, E3 +274858.291}
SPL {X  -162.820, Y  +485.759, Z    +0.000, E1   +53.138, E3 +274872.298}
ENDSPLINE

SPLINE
SPL {X  -162.820, Y  +494.645, Z    +0.000, E1   +48.544, E3 +274884.774}
ENDSPLINE

SPLINE
SPL {X  -162.820, Y  +486.578, Z    +0.000, E1   +49.194, E3 +274895.570}
SPL {X  -162.820, Y  +476.731, Z    +0.000, E1   +50.039, E3 +274907.993}
SPL {X  -162.820, Y  +466.442, Z    +0.000, E1   +50.873, E3 +274920.662}
SPL {X  -162.820, Y  +455.624, Z    +0.000, E1   +51.698, E3 +274933.733}
SPL {X  -162.820, Y  +444.568, Z    +0.000, E1   +52.608, E3 +274946.046}
SPL {X  -162.820, Y  +432.435, Z    +0.000, E1   +53.605, E3 +274958.929}
SPL {X  -162.820, Y  +419.900, Z    +0.000, E1   +54.598, E3 +274971.603}
SPL {X  -162.820, Y  +411.092, Z    +0.000, E1   +54.552, E3 +274985.123}
SPL {X  -162.820, Y  +400.244, Z    +0.000, E1   +54.630, E3 +275000.590}
SPL {X  -162.820, Y  +389.249, Z    +0.000, E1   +54.752, E3 +275016.169}
SPL {X  -162.820, Y  +380.650, Z    +0.000, E1   +54.601, E3 +275029.614}
SPL {X  -162.727, Y  +374.992, Z    +0.000, E1   +54.549, E3 +275038.296}
SPL {X  -162.216, Y  +366.490, Z    +0.000, E1   +54.549, E3 +275051.095}
SPL {X  -161.062, Y  +356.641, Z    +0.000, E1   +54.440, E3 +275066.213}
SPL {X  -159.761, Y  +349.086, Z    +0.000, E1   +54.132, E3 +275079.234}
SPL {X  -158.033, Y  +341.310, Z    +0.000, E1   +53.819, E3 +275092.624}
SPL {X  -156.195, Y  +334.528, Z    +0.000, E1   +53.534, E3 +275104.190}
SPL {X  -154.959, Y  +330.520, Z    +0.000, E1   +53.198, E3 +275111.982}
SPL {X  -152.785, Y  +324.223, Z    +0.000, E1   +52.975, E3 +275122.655}
SPL {X  -150.663, Y  +318.766, Z    +0.000, E1   +52.574, E3 +275132.688}
SPL {X  -148.923, Y  +314.679, Z    +0.000, E1   +52.172, E3 +275140.846}
SPL {X  -146.846, Y  +310.168, Z    +0.000, E1   +51.697, E3 +275149.907}
SPL {X  -140.627, Y  +298.437, Z    +0.000, E1   +54.251, E3 +275154.166}
SPL {X  -122.064, Y  +272.747, Z    +0.000, E1   +48.156, E3 +275259.692}
ENDSPLINE

SPLINE
SPL {X  -148.173, Y  +313.009, Z    +0.000, E1   +35.624, E3 +275342.737}
SPL {X  -159.343, Y  +347.032, Z    +0.000, E1   +21.245, E3 +275346.581}
SPL {X  -162.355, Y  +368.197, Z    +0.000, E1    +9.799, E3 +275347.749}
SPL {X  -162.819, Y  +380.071, Z    +0.000, E1    +2.240, E3 +275347.744}
SPL {X  -162.820, Y  +383.414, Z    +0.000, E1    -0.499, E3 +275347.707}
SPL {X  -162.820, Y  +385.887, Z    +0.000, E1    -2.819, E3 +275347.429}
SPL {X  -162.820, Y  +389.383, Z    +0.000, E1    -6.871, E3 +275347.496}
SPL {X  -162.820, Y  +393.153, Z    +0.000, E1   -11.600, E3 +275347.390}
SPL {X  -162.820, Y  +400.748, Z    +0.000, E1   -21.791, E3 +275347.181}
SPL {X  -162.820, Y  +413.615, Z    +0.000, E1   -37.560, E3 +275347.275}
SPL {X  -162.820, Y  +452.521, Z    +0.000, E1   -56.942, E3 +275361.567}
SPL {X  -162.820, Y  +459.967, Z    +0.000, E1   -57.801, E3 +275366.863}
SPL {X  -162.820, Y  +525.017, Z    +0.000, E1   -58.379, E3 +275434.982}
ENDSPLINE

SPLINE
SPL {X  -162.820, Y  +520.266, Z    +0.000, E1   -55.155, E3 +275449.474}
ENDSPLINE

SPLINE
SPL {X  -162.820, Y  +529.742, Z    +0.000, E1   -55.146, E3 +275463.190}
SPL {X  -162.820, Y  +538.383, Z    +0.000, E1   -55.306, E3 +275474.642}
SPL {X  -162.820, Y  +544.790, Z    +0.000, E1   -55.066, E3 +275485.443}
SPL {X  -162.820, Y  +555.105, Z    +0.000, E1   -55.222, E3 +275499.563}
SPL {X  -162.820, Y  +563.355, Z    +0.000, E1   -55.172, E3 +275511.630}
SPL {X  -162.820, Y  +570.590, Z    +0.000, E1   -55.270, E3 +275521.548}
SPL {X  -162.820, Y  +580.865, Z    +0.000, E1   -55.132, E3 +275537.504}
SPL {X  -162.820, Y  +591.604, Z    +0.000, E1   -55.202, E3 +275552.442}
SPL {X  -162.820, Y  +600.465, Z    +0.000, E1   -55.218, E3 +275565.230}
SPL {X  -162.820, Y  +609.951, Z    +0.000, E1   -55.211, E3 +275578.978}
SPL {X  -162.820, Y  +618.960, Z    +0.000, E1   -55.186, E3 +275592.198}
SPL {X  -162.820, Y  +627.322, Z    +0.000, E1   -55.201, E3 +275604.133}
SPL {X  -162.820, Y  +634.693, Z    +0.000, E1   -55.198, E3 +275614.850}
SPL {X  -162.820, Y  +642.452, Z    +0.000, E1   -55.141, E3 +275626.456}
SPL {X  -162.820, Y  +652.837, Z    +0.000, E1   -55.281, E3 +275640.724}
SPL {X  -162.820, Y  +660.849, Z    +0.000, E1   -55.101, E3 +275653.273}
SPL {X  -162.820, Y  +671.259, Z    +0.000, E1   -55.266, E3 +275667.569}
SPL {X  -162.498, Y  +683.731, Z    +0.000, E1   -55.157, E3 +275686.279}
SPL {X  -161.784, Y  +691.841, Z    +0.000, E1   -55.010, E3 +275698.735}
SPL {X  -160.705, Y  +699.660, Z    +0.000, E1   -54.830, E3 +275711.395}
SPL {X  -158.809, Y  +709.418, Z    +0.000, E1   -54.602, E3 +275726.867}
SPL {X  -157.115, Y  +716.223, Z    +0.000, E1   -54.227, E3 +275738.799}
SPL {X  -154.825, Y  +723.894, Z    +0.000, E1   -53.830, E3 +275752.339}
SPL {X  -152.160, Y  +731.445, Z    +0.000, E1   -53.336, E3 +275765.882}
SPL {X  -150.059, Y  +736.687, Z    +0.000, E1   -53.023, E3 +275775.047}
SPL {X  -147.746, Y  +741.922, Z    +0.000, E1   -52.631, E3 +275784.755}
SPL {X  -144.373, Y  +748.778, Z    +0.000, E1   -52.887, E3 +275793.168}
SPL {X  -137.947, Y  +759.993, Z    +0.000, E1   -55.381, E3 +275796.277}
SPL {X  -123.111, Y  +780.056, Z    +0.000, E1   -48.144, E3 +275895.413}
ENDSPLINE

